KUKA KRL program: MyProgram_297().src

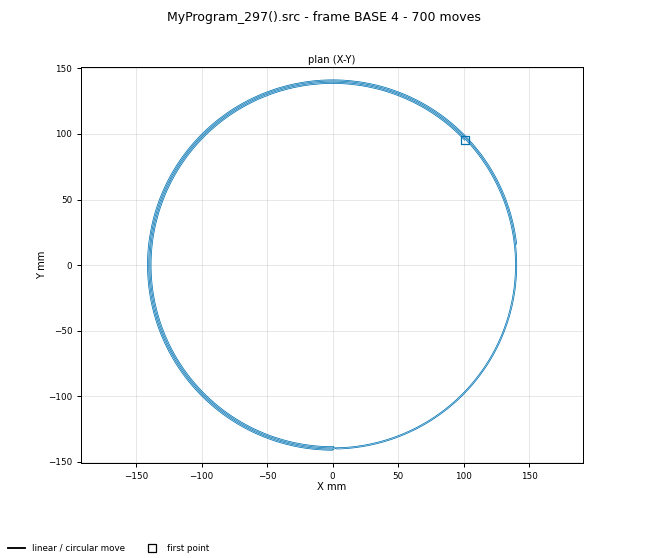
[picture p0: tool path of MyProgram_297().src in frame BASE 4, 700 of 700 moves have a stored position in this frame; points joined in program order, loops and branches not executed]
&ACCESS RVP
&REL 1
&PARAM TEMPLATE = C:\KRC\Roboter\Template\vorgabe
&PARAM EDITMASK = *
DEF MyProgram_297()
; ---- Setting reference (Base) ----
$BASE = BASE_DATA[4]

; --------------------------
; ---- Setting tool (TCP) ----
$TOOL = TOOL_DATA[3]
; --------------------------

$VEL.CP = VEL_APROX_PRINT
Startdeposition()
$VEL.CP = VEL_PRINT
LIN {X 100.7253,Y 95.1993,Z 178,A 45.1917,B 6.1181,C 0.1489,E1 6.2362,E2 407.2014} C_DIS
LIN {X 97.6837,Y 98.3177,Z 178,A 47.1151,B 6.1182,C 0.1434,E1 6.2323,E2 405.262} C_DIS
LIN {X 93.7907,Y 102.0381,Z 178,A 49.1623,B 6.1182,C 0.1418,E1 6.2282,E2 403.237} C_DIS
LIN {X 90.4705,Y 104.9931,Z 178,A 50.9851,B 6.1183,C 0.1386,E1 6.2244,E2 401.4158} C_DIS
LIN {X 87.1947,Y 107.7293,Z 178,A 52.6581,B 6.1183,C 0.1368,E1 6.2208,E2 399.754} C_DIS
LIN {X 83.9283,Y 110.2933,Z 178,A 54.4404,B 6.1185,C 0.1327,E1 6.2168,E2 397.9633} C_DIS
LIN {X 80.2806,Y 112.9764,Z 178,A 57.0009,B 6.1188,C 0.119,E1 6.2108,E2 395.3153} C_DIS
LIN {X 75.162,Y 116.444,Z 178,A 58.6179,B 6.1185,C 0.1293,E1 6.2073,E2 393.8171} C_DIS
LIN {X 71.7588,Y 118.5713,Z 178,A 60.415,B 6.1186,C 0.1247,E1 6.203,E2 392.0026} C_DIS
LIN {X 67.9906,Y 120.7715,Z 178,A 62.2218,B 6.1186,C 0.1221,E1 6.1986,E2 390.1954} C_DIS
LIN {X 64.2773,Y 122.7858,Z 178,A 63.932,B 6.1187,C 0.1203,E1 6.1944,E2 388.4897} C_DIS
LIN {X 60.7829,Y 124.554,Z 178,A 66.1002,B 6.1189,C 0.11,E1 6.1888,E2 386.2523} C_DIS
LIN {X 56.039,Y 126.7593,Z 178,A 67.8115,B 6.1189,C 0.1142,E1 6.1846,E2 384.5984} C_DIS
LIN {X 52.6665,Y 128.1983,Z 178,A 69.1021,B 6.1189,C 0.1158,E1 6.1813,E2 383.3363} C_DIS
LIN {X 50.1247,Y 129.2109,Z 178,A 70.2479,B 6.1189,C 0.1144,E1 6.1784,E2 382.1887} C_DIS
LIN {X 46.6313,Y 130.5129,Z 178,A 71.7515,B 6.1189,C 0.1134,E1 6.1744,E2 380.6901} C_DIS
LIN {X 43.0422,Y 131.7419,Z 178,A 73.3054,B 6.1189,C 0.1121,E1 6.1703,E2 379.1383} C_DIS
LIN {X 40.2799,Y 132.6106,Z 178,A 74.5276,B 6.1189,C 0.1107,E1 6.167,E2 377.9131} C_DIS
LIN {X 37.0505,Y 133.5489,Z 178,A 75.904,B 6.1189,C 0.1098,E1 6.1633,E2 376.5387} C_DIS
LIN {X 32.881,Y 134.6365,Z 178,A 77.8166,B 6.1189,C 0.1067,E1 6.1581,E2 374.6101} C_DIS
LIN {X 25.5972,Y 136.2093,Z 178,A 80.8088,B 6.1189,C 0.1061,E1 6.15,E2 371.6299} C_DIS
LIN {X 21.3585,Y 136.9374,Z 178,A 83.4736,B 6.1192,C 0.0929,E1 6.1423,E2 368.8539} C_DIS
LIN {X 14.2754,Y 137.857,Z 178,A 85.3447,B 6.119,C 0.1068,E1 6.1375,E2 367.1202} C_DIS
LIN {X 9.967,Y 138.2343,Z 178,A 87.2432,B 6.119,C 0.1048,E1 6.1322,E2 365.2086} C_DIS
LIN {X 6.2445,Y 138.4543,Z 178,A 88.9169,B 6.119,C 0.1028,E1 6.1275,E2 363.5191} C_DIS
LIN {X 1.7423,Y 138.5834,Z 178,A 90.7344,B 6.119,C 0.1032,E1 6.1224,E2 361.7079} C_DIS
LIN {X -2.2127,Y 138.5756,Z 178,A 92.2544,B 6.119,C 0.1048,E1 6.1182,E2 360.2029} C_DIS
LIN {X -5.8911,Y 138.4688,Z 178,A 93.7442,B 6.119,C 0.1053,E1 6.114,E2 358.7178} C_DIS
LIN {X -9.6122,Y 138.2602,Z 178,A 95.28,B 6.119,C 0.1056,E1 6.1098,E2 357.1834} C_DIS
LIN {X -18.0083,Y 137.4181,Z 178,A 98.4994,B 6.119,C 0.1101,E1 6.101,E2 353.9995} C_DIS
LIN {X -22.9135,Y 136.6857,Z 178,A 100.7104,B 6.119,C 0.1088,E1 6.0948,E2 351.7697} C_DIS
LIN {X -26.0665,Y 136.1196,Z 178,A 102.2509,B 6.119,C 0.1067,E1 6.0905,E2 350.2031} C_DIS
LIN {X -29.2745,Y 135.4658,Z 178,A 103.6444,B 6.119,C 0.107,E1 6.0866,E2 348.8054} C_DIS
LIN {X -33.7927,Y 134.4103,Z 178,A 105.6072,B 6.119,C 0.1077,E1 6.0813,E2 346.8383} C_DIS
LIN {X -37.8957,Y 133.3125,Z 178,A 107.194,B 6.119,C 0.1111,E1 6.0771,E2 345.2736} C_DIS
LIN {X -40.7847,Y 132.4561,Z 178,A 108.5376,B 6.119,C 0.1109,E1 6.0735,E2 343.9187} C_DIS
LIN {X -44.1224,Y 131.3822,Z 178,A 109.9811,B 6.1189,C 0.1122,E1 6.0696,E2 342.4769} C_DIS
LIN {X -48.0912,Y 129.9826,Z 178,A 111.7643,B 6.1189,C 0.1133,E1 6.0649,E2 340.6895} C_DIS
LIN {X -55.095,Y 127.171,Z 178,A 114.518,B 6.1187,C 0.1211,E1 6.058,E2 337.9836} C_DIS
LIN {X -58.8642,Y 125.4731,Z 178,A 116.9315,B 6.1188,C 0.1146,E1 6.0516,E2 335.4838} C_DIS
LIN {X -62.0184,Y 123.9445,Z 178,A 118.0563,B 6.1188,C 0.1203,E1 6.0489,E2 334.4006} C_DIS
LIN {X -64.646,Y 122.5922,Z 178,A 119.2808,B 6.1188,C 0.1219,E1 6.0459,E2 333.1766} C_DIS
LIN {X -68.3234,Y 120.5842,Z 178,A 121.1678,B 6.1187,C 0.1224,E1 6.0412,E2 331.2716} C_DIS
LIN {X -72.2248,Y 118.2883,Z 178,A 123.0723,B 6.1187,C 0.1248,E1 6.0366,E2 329.3644} C_DIS
LIN {X -76.1855,Y 115.7767,Z 178,A 125.0168,B 6.1186,C 0.1277,E1 6.0321,E2 327.4208} C_DIS
LIN {X -80.0632,Y 113.13,Z 178,A 127.0679,B 6.1186,C 0.1296,E1 6.0274,E2 325.3575} C_DIS
LIN {X -83.5881,Y 110.551,Z 178,A 128.8041,B 6.1185,C 0.1334,E1 6.0235,E2 323.6315} C_DIS
LIN {X -86.8755,Y 107.9868,Z 178,A 130.5701,B 6.1185,C 0.136,E1 6.0196,E2 321.8616} C_DIS
LIN {X -90.4313,Y 105.0269,Z 178,A 132.5625,B 6.1183,C 0.1386,E1 6.0154,E2 319.8609} C_DIS
LIN {X -94.299,Y 101.5687,Z 178,A 134.5455,B 6.1183,C 0.1446,E1 6.0113,E2 317.8999} C_DIS
LIN {X -97.1107,Y 98.8837,Z 178,A 136.3105,B 6.1182,C 0.146,E1 6.0077,E2 316.1166} C_DIS
LIN {X -100.4054,Y 95.537,Z 178,A 138.3895,B 6.1182,C 0.1484,E1 6.0037,E2 314.0221} C_DIS
LIN {X -103.4582,Y 92.2224,Z 178,A 140.1155,B 6.118,C 0.1539,E1 6.0005,E2 312.3149} C_DIS
LIN {X -106.0375,Y 89.2444,Z 178,A 141.7656,B 6.1179,C 0.1572,E1 5.9975,E2 310.6635} C_DIS
LIN {X -108.3675,Y 86.4,Z 178,A 143.3929,B 6.1179,C 0.1594,E1 5.9946,E2 309.0241} C_DIS
LIN {X -111.3703,Y 82.4939,Z 178,A 145.4041,B 6.1177,C 0.1643,E1 5.9912,E2 307.018} C_DIS
LIN {X -113.712,Y 79.2342,Z 178,A 147.1609,B 6.1177,C 0.1671,E1 5.9884,E2 305.2505} C_DIS
LIN {X -116.3293,Y 75.3392,Z 178,A 149.1049,B 6.1175,C 0.1717,E1 5.9854,E2 303.3076} C_DIS
LIN {X -118.5224,Y 71.8397,Z 178,A 150.8723,B 6.1175,C 0.1752,E1 5.9828,E2 301.5343} C_DIS
LIN {X -120.7551,Y 68.0198,Z 178,A 152.7493,B 6.1173,C 0.1793,E1 5.9802,E2 299.6529} C_DIS
LIN {X -123.7351,Y 62.4322,Z 178,A 155.3187,B 6.1171,C 0.1864,E1 5.9768,E2 297.092} C_DIS
LIN {X -125.4863,Y 58.8358,Z 178,A 156.9727,B 6.117,C 0.1907,E1 5.9748,E2 295.4395} C_DIS
LIN {X -126.4956,Y 56.6285,Z 178,A 158.0829,B 6.117,C 0.1922,E1 5.9736,E2 294.3167} C_DIS
LIN {X -127.9618,Y 53.2329,Z 178,A 160.2866,B 6.117,C 0.1891,E1 5.9711,E2 292.0288} C_DIS
LIN {X -129.9199,Y 48.2586,Z 178,A 162.2344,B 6.1167,C 0.1978,E1 5.9692,E2 290.1164} C_DIS
LIN {X -131.1832,Y 44.7149,Z 178,A 163.4264,B 6.1165,C 0.2058,E1 5.9682,E2 288.972} C_DIS
LIN {X -132.0421,Y 42.1053,Z 178,A 164.6413,B 6.1164,C 0.2081,E1 5.9671,E2 287.748} C_DIS
LIN {X -133.1106,Y 38.5962,Z 178,A 166.1683,B 6.1162,C 0.2121,E1 5.9659,E2 286.2209} C_DIS
LIN {X -134.175,Y 34.7196,Z 178,A 167.7959,B 6.1161,C 0.2171,E1 5.9648,E2 284.5993} C_DIS
LIN {X -134.8127,Y 32.1502,Z 178,A 168.9852,B 6.1161,C 0.2192,E1 5.964,E2 283.3989} C_DIS
LIN {X -135.5798,Y 28.7468,Z 178,A 170.8753,B 6.1161,C 0.2185,E1 5.9628,E2 281.4531} C_DIS
LIN {X -136.3289,Y 24.9548,Z 178,A 171.9926,B 6.1157,C 0.228,E1 5.9623,E2 280.3983} C_DIS
LIN {X -137.035,Y 20.7283,Z 178,A 173.8658,B 6.1155,C 0.232,E1 5.9614,E2 278.5138} C_DIS
LIN {X -137.4731,Y 17.5883,Z 178,A 175.2734,B 6.1155,C 0.2347,E1 5.9609,E2 277.0949} C_DIS
LIN {X -138.0078,Y 12.7341,Z 178,A 177.5784,B 6.1153,C 0.2374,E1 5.9603,E2 274.7552} C_DIS
LIN {X -138.3575,Y 8.0894,Z 178,A 179.3067,B 6.115,C 0.245,E1 5.9599,E2 273.0537} C_DIS
LIN {X -138.5482,Y 3.5444,Z 178,A -178.763,B 6.1148,C 0.2499,E1 5.9597,E2 271.1185} C_DIS
LIN {X -138.588,Y -1.3629,Z 178,A -176.4182,B 6.1148,C 0.2524,E1 5.9597,E2 268.7351} C_DIS
LIN {X -138.4345,Y -6.6374,Z 178,A -174.403,B 6.1144,C 0.2603,E1 5.96,E2 266.7428} C_DIS
LIN {X -138.1855,Y -10.6361,Z 178,A -172.6569,B 6.1142,C 0.2641,E1 5.9603,E2 264.9864} C_DIS
LIN {X -137.7888,Y -14.9093,Z 178,A -170.8181,B 6.114,C 0.2684,E1 5.9608,E2 263.1406} C_DIS
LIN {X -137.3126,Y -18.8119,Z 178,A -169.1039,B 6.1139,C 0.2721,E1 5.9615,E2 261.4163} C_DIS
LIN {X -136.7527,Y -22.5121,Z 178,A -167.6567,B 6.1136,C 0.2775,E1 5.9621,E2 259.983} C_DIS
LIN {X -136.1286,Y -26.0195,Z 178,A -166.1799,B 6.1135,C 0.2816,E1 5.9628,E2 258.5067} C_DIS
LIN {X -135.4008,Y -29.5757,Z 178,A -164.6551,B 6.1133,C 0.2855,E1 5.9637,E2 256.9798} C_DIS
LIN {X -134.6153,Y -32.9689,Z 178,A -163.1742,B 6.1131,C 0.289,E1 5.9647,E2 255.4947} C_DIS
LIN {X -133.8465,Y -35.9606,Z 178,A -161.9285,B 6.1129,C 0.2929,E1 5.9656,E2 254.2538} C_DIS
LIN {X -133.0131,Y -38.9292,Z 178,A -160.4892,B 6.1129,C 0.2946,E1 5.9667,E2 252.7941} C_DIS
LIN {X -131.8935,Y -42.5703,Z 178,A -158.855,B 6.1127,C 0.2982,E1 5.9681,E2 251.1534} C_DIS
LIN {X -130.1182,Y -47.7261,Z 178,A -156.6629,B 6.1123,C 0.3049,E1 5.9701,E2 248.9706} C_DIS
LIN {X -128.9024,Y -50.9183,Z 178,A -155.2152,B 6.1122,C 0.3082,E1 5.9716,E2 247.5191} C_DIS
LIN {X -127.6594,Y -53.9569,Z 178,A -153.8291,B 6.112,C 0.3115,E1 5.9731,E2 246.1301} C_DIS
LIN {X -126.4571,Y -56.7145,Z 178,A -152.4951,B 6.1119,C 0.3137,E1 5.9746,E2 244.7851} C_DIS
LIN {X -124.9377,Y -59.988,Z 178,A -150.9958,B 6.1117,C 0.3174,E1 5.9764,E2 243.2856} C_DIS
LIN {X -123.1323,Y -63.6163,Z 178,A -148.8755,B 6.1117,C 0.3167,E1 5.9792,E2 241.1085} C_DIS
LIN {X -121.2539,Y -67.1265,Z 178,A -147.9414,B 6.1111,C 0.3287,E1 5.9803,E2 240.2674} C_DIS
LIN {X -118.7782,Y -71.4166,Z 178,A -145.3999,B 6.1111,C 0.3281,E1 5.9839,E2 237.663} C_DIS
LIN {X -116.3136,Y -75.3634,Z 178,A -143.4433,B 6.1109,C 0.3323,E1 5.9869,E2 235.703} C_DIS
LIN {X -113.931,Y -78.9194,Z 178,A -141.6395,B 6.1107,C 0.336,E1 5.9897,E2 233.8955} C_DIS
LIN {X -111.2363,Y -82.6739,Z 178,A -139.711,B 6.1105,C 0.3401,E1 5.9929,E2 231.9653} C_DIS
LIN {X -108.3847,Y -86.3785,Z 178,A -137.7678,B 6.1103,C 0.3442,E1 5.9963,E2 230.0215} C_DIS
LIN {X -105.5981,Y -89.7636,Z 178,A -135.914,B 6.1101,C 0.3476,E1 5.9996,E2 228.1629} C_DIS
LIN {X -102.6518,Y -93.1187,Z 178,A -134.0717,B 6.1098,C 0.3515,E1 6.003,E2 226.3216} C_DIS
LIN {X -99.832,Y -96.1362,Z 178,A -132.2581,B 6.1098,C 0.3536,E1 6.0065,E2 224.4945} C_DIS
LIN {X -96.606,Y -99.3772,Z 178,A -130.4005,B 6.1095,C 0.3577,E1 6.0102,E2 222.6417} C_DIS
LIN {X -93.4399,Y -102.3603,Z 178,A -128.5488,B 6.1093,C 0.3604,E1 6.014,E2 220.7834} C_DIS
LIN {X -90.146,Y -105.2726,Z 178,A -126.6642,B 6.1092,C 0.3629,E1 6.018,E2 218.8903} C_DIS
LIN {X -86.5888,Y -108.2173,Z 178,A -124.7614,B 6.109,C 0.3662,E1 6.0221,E2 216.9886} C_DIS
LIN {X -83.0471,Y -110.9584,Z 178,A -122.3531,B 6.1092,C 0.3625,E1 6.0277,E2 214.5073} C_DIS
LIN {X -78.8969,Y -113.9467,Z 178,A -120.9727,B 6.1085,C 0.3748,E1 6.0306,E2 213.2236} C_DIS
LIN {X -76.2379,Y -115.7422,Z 178,A -119.2641,B 6.1086,C 0.372,E1 6.0347,E2 211.465} C_DIS
LIN {X -71.9067,Y -118.4818,Z 178,A -117.2397,B 6.1084,C 0.3762,E1 6.0395,E2 209.453} C_DIS
LIN {X -67.9145,Y -120.8143,Z 178,A -115.3273,B 6.1082,C 0.3787,E1 6.0441,E2 207.5406} C_DIS
LIN {X -63.9131,Y -122.9771,Z 178,A -112.8863,B 6.1085,C 0.3739,E1 6.0503,E2 205.0255} C_DIS
LIN {X -59.3138,Y -125.2598,Z 178,A -111.7959,B 6.1076,C 0.3895,E1 6.0527,E2 204.0707} C_DIS
LIN {X -55.6661,Y -126.9241,Z 178,A -109.7533,B 6.1077,C 0.3864,E1 6.0581,E2 201.9778} C_DIS
LIN {X -52.0497,Y -128.4477,Z 178,A -108.0497,B 6.1077,C 0.3869,E1 6.0625,E2 200.2632} C_DIS
LIN {X -48.7938,Y -129.7195,Z 178,A -106.5077,B 6.1077,C 0.3869,E1 6.0665,E2 198.7082} C_DIS
LIN {X -45.3055,Y -130.9785,Z 178,A -105.0417,B 6.1076,C 0.3891,E1 6.0704,E2 197.2509} C_DIS
LIN {X -41.5118,Y -132.2316,Z 178,A -103.4267,B 6.1075,C 0.3909,E1 6.0747,E2 195.6404} C_DIS
LIN {X -38.64,Y -133.0978,Z 178,A -102.1278,B 6.1075,C 0.3909,E1 6.0782,E2 194.3334} C_DIS
LIN {X -33.1805,Y -134.5643,Z 178,A -99.0562,B 6.108,C 0.3825,E1 6.0867,E2 191.164} C_DIS
LIN {X -27.5769,Y -135.8216,Z 178,A -97.6586,B 6.1071,C 0.3968,E1 6.0902,E2 189.8949} C_DIS
LIN {X -21.1122,Y -136.9755,Z 178,A -94.6575,B 6.1073,C 0.3939,E1 6.0986,E2 186.8554} C_DIS
LIN {X -17.645,Y -137.4657,Z 178,A -93.3149,B 6.1072,C 0.3958,E1 6.1023,E2 185.5262} C_DIS
LIN {X -14.6413,Y -137.8176,Z 178,A -91.9734,B 6.1072,C 0.3947,E1 6.106,E2 184.1721} C_DIS
LIN {X -10.2752,Y -138.2118,Z 178,A -90.1388,B 6.1072,C 0.3947,E1 6.1111,E2 182.3339} C_DIS
LIN {X -6.937,Y -138.4194,Z 178,A -88.7327,B 6.1072,C 0.3944,E1 6.1151,E2 180.9242} C_DIS
LIN {X -3.2907,Y -138.5553,Z 178,A -87.2392,B 6.1072,C 0.3945,E1 6.1192,E2 179.4319} C_DIS
LIN {X 1.0123,Y -138.5881,Z 178,A -85.629,B 6.1071,C 0.3967,E1 6.1237,E2 177.8431} C_DIS
Enddeposition()
LIN {X 1.0123,Y -138.5881,Z 178,A -85.629,B 6.1071,C 0.3967,E1 6.1237,E2 177.8431} C_DIS
Startdeposition()
$VEL.CP = VEL_PRINT
LIN {X 0.3223,Y -139.4978,Z 178,A -86.4941,B 6.0436,C 0.4078,E1 6.0583,E2 178.8356} C_DIS
LIN {X -3.5454,Y -139.4527,Z 178,A -87.9992,B 6.0436,C 0.4067,E1 6.0541,E2 180.3305} C_DIS
LIN {X -7.1717,Y -139.313,Z 178,A -89.4579,B 6.0437,C 0.4063,E1 6.05,E2 181.7857} C_DIS
LIN {X -10.8678,Y -139.0752,Z 178,A -91.0003,B 6.0437,C 0.4064,E1 6.0457,E2 183.3315} C_DIS
LIN {X -14.386,Y -138.7546,Z 178,A -92.4328,B 6.0437,C 0.406,E1 6.0417,E2 184.7622} C_DIS
LIN {X -18.0156,Y -138.3291,Z 178,A -93.9271,B 6.0437,C 0.4055,E1 6.0376,E2 186.2561} C_DIS
LIN {X -21.615,Y -137.8127,Z 178,A -95.4504,B 6.0437,C 0.4055,E1 6.0334,E2 187.7838} C_DIS
LIN {X -26.509,Y -136.9556,Z 178,A -97.5705,B 6.0437,C 0.4057,E1 6.0275,E2 189.915} C_DIS
LIN {X -31.0309,Y -136.0019,Z 178,A -99.4007,B 6.0439,C 0.4039,E1 6.0225,E2 191.7368} C_DIS
LIN {X -35.1536,Y -134.997,Z 178,A -101.3758,B 6.0437,C 0.4059,E1 6.0171,E2 193.7428} C_DIS
LIN {X -40.222,Y -133.5739,Z 178,A -103.4323,B 6.0439,C 0.4031,E1 6.0116,E2 195.7859} C_DIS
LIN {X -44.3434,Y -132.2617,Z 178,A -105.0412,B 6.0442,C 0.3996,E1 6.0074,E2 197.3732} C_DIS
LIN {X -47.3233,Y -131.2246,Z 178,A -106.5007,B 6.0441,C 0.4006,E1 6.0035,E2 198.8544} C_DIS
LIN {X -51.8194,Y -129.5155,Z 178,A -108.3865,B 6.0443,C 0.3976,E1 5.9986,E2 200.7287} C_DIS
LIN {X -54.7237,Y -128.3167,Z 178,A -109.8416,B 6.0443,C 0.3984,E1 5.9948,E2 202.2056} C_DIS
LIN {X -58.9864,Y -126.4129,Z 178,A -111.6098,B 6.0445,C 0.3944,E1 5.9904,E2 203.9543} C_DIS
LIN {X -62.6068,Y -124.6596,Z 178,A -113.4277,B 6.0445,C 0.3946,E1 5.9858,E2 205.7941} C_DIS
LIN {X -66.4871,Y -122.6357,Z 178,A -115.242,B 6.0446,C 0.3926,E1 5.9813,E2 207.6107} C_DIS
LIN {X -70.5308,Y -120.3551,Z 178,A -117.1397,B 6.0448,C 0.3899,E1 5.9767,E2 209.5071} C_DIS
LIN {X -74.4572,Y -117.9663,Z 178,A -118.9485,B 6.045,C 0.3863,E1 5.9724,E2 211.3056} C_DIS
LIN {X -77.8084,Y -115.7841,Z 178,A -120.8356,B 6.045,C 0.3868,E1 5.968,E2 213.2245} C_DIS
LIN {X -83.4625,Y -111.7764,Z 178,A -123.5507,B 6.0454,C 0.3808,E1 5.9619,E2 215.9223} C_DIS
LIN {X -86.935,Y -109.0974,Z 178,A -125.404,B 6.0455,C 0.3784,E1 5.9578,E2 217.782} C_DIS
LIN {X -90.4421,Y -106.2081,Z 178,A -127.2994,B 6.0457,C 0.3754,E1 5.9537,E2 219.6809} C_DIS
LIN {X -93.8098,Y -103.2456,Z 178,A -129.1509,B 6.0459,C 0.3722,E1 5.9498,E2 221.5333} C_DIS
LIN {X -97.0198,Y -100.2351,Z 178,A -130.9882,B 6.0461,C 0.3691,E1 5.9461,E2 223.3741} C_DIS
LIN {X -100.0855,Y -97.1744,Z 178,A -132.8486,B 6.0462,C 0.3665,E1 5.9424,E2 225.2445} C_DIS
LIN {X -103.3151,Y -93.7332,Z 178,A -134.7654,B 6.0465,C 0.3624,E1 5.9388,E2 227.158} C_DIS
LIN {X -106.1489,Y -90.5118,Z 178,A -136.5955,B 6.0467,C 0.3594,E1 5.9355,E2 228.9964} C_DIS
LIN {X -108.9179,Y -87.1606,Z 178,A -138.4497,B 6.0468,C 0.3564,E1 5.9322,E2 230.8589} C_DIS
LIN {X -111.7183,Y -83.5405,Z 178,A -140.3561,B 6.0471,C 0.3525,E1 5.9289,E2 232.7681} C_DIS
LIN {X -114.4517,Y -79.7544,Z 178,A -142.2746,B 6.0473,C 0.3481,E1 5.9258,E2 234.686} C_DIS
LIN {X -116.2615,Y -77.0934,Z 178,A -143.7509,B 6.0473,C 0.3468,E1 5.9235,E2 236.1817} C_DIS
LIN {X -118.9476,Y -72.8794,Z 178,A -145.6851,B 6.0477,C 0.3406,E1 5.9207,E2 238.0996} C_DIS
LIN {X -120.3674,Y -70.51,Z 178,A -147.2646,B 6.0477,C 0.3427,E1 5.9184,E2 239.7359} C_DIS
LIN {X -122.4618,Y -66.8059,Z 178,A -148.8201,B 6.048,C 0.3363,E1 5.9163,E2 241.2659} C_DIS
LIN {X -124.8761,Y -62.1739,Z 178,A -150.8063,B 6.0484,C 0.3292,E1 5.9138,E2 243.2305} C_DIS
LIN {X -126.4932,Y -58.8126,Z 178,A -152.5062,B 6.0484,C 0.3271,E1 5.9118,E2 244.9512} C_DIS
LIN {X -128.5303,Y -54.2179,Z 178,A -154.363,B 6.0489,C 0.3196,E1 5.9097,E2 246.7802} C_DIS
LIN {X -129.8442,Y -50.9913,Z 178,A -156.0907,B 6.0489,C 0.319,E1 5.9079,E2 248.5452} C_DIS
LIN {X -131.9966,Y -45.1295,Z 178,A -158.5339,B 6.0493,C 0.3108,E1 5.9056,E2 250.9713} C_DIS
LIN {X -133.1589,Y -41.5781,Z 178,A -160.1436,B 6.0495,C 0.3075,E1 5.9042,E2 252.5897} C_DIS
LIN {X -134.1836,Y -38.1385,Z 178,A -161.6845,B 6.0497,C 0.3042,E1 5.903,E2 254.1382} C_DIS
LIN {X -135.1933,Y -34.3833,Z 178,A -163.248,B 6.0499,C 0.2994,E1 5.9019,E2 255.6963} C_DIS
LIN {X -135.975,Y -31.149,Z 178,A -164.651,B 6.0501,C 0.296,E1 5.901,E2 257.1031} C_DIS
LIN {X -136.7965,Y -27.3206,Z 178,A -166.3624,B 6.0503,C 0.2926,E1 5.9001,E2 258.8265} C_DIS
LIN {X -137.5642,Y -23.1428,Z 178,A -167.8976,B 6.0506,C 0.2856,E1 5.8993,E2 260.3337} C_DIS
LIN {X -138.0283,Y -20.1962,Z 178,A -169.3041,B 6.0506,C 0.284,E1 5.8987,E2 261.7625} C_DIS
LIN {X -138.5928,Y -15.8732,Z 178,A -171.649,B 6.0506,C 0.2847,E1 5.8979,E2 264.1765} C_DIS
LIN {X -139.0057,Y -11.701,Z 178,A -172.9455,B 6.0511,C 0.2754,E1 5.8976,E2 265.4177} C_DIS
LIN {X -139.2898,Y -7.6336,Z 178,A -175.258,B 6.051,C 0.2772,E1 5.8972,E2 267.8098} C_DIS
LIN {X -139.4717,Y -2.7059,Z 178,A -177.3632,B 6.0512,C 0.2722,E1 5.8972,E2 269.9234} C_DIS
LIN {X -139.4768,Y 2.4022,Z 178,A -178.8572,B 6.0517,C 0.26,E1 5.8972,E2 271.3395} C_DIS
LIN {X -139.365,Y 6.1135,Z 178,A 178.8526,B 6.0516,C 0.2635,E1 5.8975,E2 273.725} C_DIS
LIN {X -139.0193,Y 11.54,Z 178,A 176.7976,B 6.0519,C 0.2553,E1 5.8979,E2 275.7558} C_DIS
LIN {X -138.5925,Y 15.8752,Z 178,A 175.3404,B 6.0523,C 0.2468,E1 5.8983,E2 277.1697} C_DIS
LIN {X -138.1322,Y 19.4689,Z 178,A 173.8745,B 6.0525,C 0.2424,E1 5.8989,E2 278.6316} C_DIS
LIN {X -137.5997,Y 22.9302,Z 178,A 172.3164,B 6.0525,C 0.2395,E1 5.8996,E2 280.2035} C_DIS
LIN {X -136.4381,Y 29.0561,Z 178,A 169.918,B 6.0529,C 0.2307,E1 5.9009,E2 282.5792} C_DIS
LIN {X -135.7528,Y 32.1087,Z 178,A 168.4295,B 6.0529,C 0.2292,E1 5.9018,E2 284.0923} C_DIS
LIN {X -134.7915,Y 35.926,Z 178,A 166.852,B 6.0532,C 0.2243,E1 5.9029,E2 285.6634} C_DIS
LIN {X -134.0376,Y 38.6482,Z 178,A 165.6447,B 6.0532,C 0.2216,E1 5.9038,E2 286.8756} C_DIS
LIN {X -132.9994,Y 42.0799,Z 178,A 164.0526,B 6.0534,C 0.2188,E1 5.9051,E2 288.4815} C_DIS
LIN {X -131.9971,Y 45.1279,Z 178,A 162.9028,B 6.0535,C 0.2135,E1 5.9061,E2 289.609} C_DIS
LIN {X -130.7766,Y 48.5494,Z 178,A 161.4479,B 6.0537,C 0.2091,E1 5.9075,E2 291.0579} C_DIS
LIN {X -129.7175,Y 51.3141,Z 178,A 159.7641,B 6.0537,C 0.2107,E1 5.9093,E2 292.7993} C_DIS
LIN {X -127.6546,Y 56.2518,Z 178,A 157.6571,B 6.0539,C 0.204,E1 5.9116,E2 294.893} C_DIS
LIN {X -126.1299,Y 59.5901,Z 178,A 156.3412,B 6.0541,C 0.1981,E1 5.9131,E2 296.1835} C_DIS
LIN {X -124.2884,Y 63.3384,Z 178,A 154.1697,B 6.0541,C 0.1984,E1 5.9159,E2 298.4105} C_DIS
LIN {X -122.6034,Y 66.5464,Z 178,A 152.8451,B 6.0542,C 0.193,E1 5.9176,E2 299.7134} C_DIS
LIN {X -120.4136,Y 70.4314,Z 178,A 150.9757,B 6.0544,C 0.1888,E1 5.9202,E2 301.5859} C_DIS
LIN {X -117.9566,Y 74.4727,Z 178,A 149.0545,B 6.0545,C 0.1839,E1 5.923,E2 303.5026} C_DIS
LIN {X -115.5646,Y 78.133,Z 178,A 147.2061,B 6.0546,C 0.1801,E1 5.9259,E2 305.356} C_DIS
LIN {X -113.0534,Y 81.7244,Z 178,A 145.4324,B 6.0548,C 0.1757,E1 5.9288,E2 307.1248} C_DIS
LIN {X -109.9842,Y 85.8114,Z 178,A 143.179,B 6.0548,C 0.1726,E1 5.9326,E2 309.3956} C_DIS
LIN {X -107.16,Y 89.3133,Z 178,A 141.3302,B 6.055,C 0.1685,E1 5.9359,E2 311.2429} C_DIS
LIN {X -103.6159,Y 93.4013,Z 178,A 138.6156,B 6.055,C 0.1691,E1 5.941,E2 314.0166} C_DIS
LIN {X -100.4507,Y 96.7971,Z 178,A 137.0856,B 6.0552,C 0.161,E1 5.9439,E2 315.4983} C_DIS
LIN {X -97.3979,Y 99.8686,Z 178,A 134.8234,B 6.0552,C 0.1628,E1 5.9485,E2 317.8188} C_DIS
LIN {X -93.8656,Y 103.195,Z 178,A 132.8703,B 6.0552,C 0.1585,E1 5.9525,E2 319.7653} C_DIS
LIN {X -90.4971,Y 106.1613,Z 178,A 131.396,B 6.0554,C 0.151,E1 5.9556,E2 321.1923} C_DIS
LIN {X -86.4274,Y 109.5004,Z 178,A 129.0822,B 6.0554,C 0.1488,E1 5.9606,E2 323.5231} C_DIS
LIN {X -80.5402,Y 113.9001,Z 178,A 126.1633,B 6.0556,C 0.1427,E1 5.9672,E2 326.4272} C_DIS
LIN {X -76.9222,Y 116.3743,Z 178,A 124.3085,B 6.0556,C 0.1404,E1 5.9715,E2 328.2873} C_DIS
LIN {X -72.9661,Y 118.8944,Z 178,A 122.3976,B 6.0557,C 0.1373,E1 5.976,E2 330.1948} C_DIS
LIN {X -69.0331,Y 121.2204,Z 178,A 120.4994,B 6.0557,C 0.1349,E1 5.9806,E2 332.0941} C_DIS
LIN {X -65.2642,Y 123.2889,Z 178,A 118.7277,B 6.0559,C 0.1326,E1 5.9849,E2 333.8652} C_DIS
LIN {X -62.4865,Y 124.7219,Z 178,A 117.2552,B 6.0559,C 0.1332,E1 5.9887,E2 335.3602} C_DIS
LIN {X -57.55,Y 127.074,Z 178,A 115.2692,B 6.0559,C 0.1275,E1 5.9936,E2 337.3123} C_DIS
LIN {X -52.8703,Y 129.0919,Z 178,A 112.7558,B 6.0559,C 0.1302,E1 6.0002,E2 339.8763} C_DIS
LIN {X -49.5221,Y 130.4123,Z 178,A 111.5938,B 6.056,C 0.1249,E1 6.0031,E2 340.9981} C_DIS
LIN {X -45.9172,Y 131.7235,Z 178,A 110.043,B 6.056,C 0.1231,E1 6.0072,E2 342.5447} C_DIS
LIN {X -42.5902,Y 132.8364,Z 178,A 108.6703,B 6.056,C 0.1211,E1 6.0108,E2 343.9079} C_DIS
LIN {X -39.2866,Y 133.8506,Z 178,A 107.219,B 6.0561,C 0.1203,E1 6.0147,E2 345.3623} C_DIS
LIN {X -34.7857,Y 135.0912,Z 178,A 105.1925,B 6.0561,C 0.1203,E1 6.0202,E2 347.4011} C_DIS
LIN {X -31.2494,Y 135.952,Z 178,A 103.7489,B 6.0561,C 0.1187,E1 6.0241,E2 348.8374} C_DIS
LIN {X -27.7276,Y 136.7137,Z 178,A 102.1669,B 6.0561,C 0.1191,E1 6.0285,E2 350.4313} C_DIS
LIN {X -19.1379,Y 138.1795,Z 178,A 98.6078,B 6.0561,C 0.1173,E1 6.0383,E2 353.986} C_DIS
LIN {X -16,Y 138.5777,Z 178,A 96.7185,B 6.0561,C 0.1245,E1 6.0437,E2 355.9474} C_DIS
LIN {X -10.874,Y 139.0747,Z 178,A 95.1928,B 6.0561,C 0.1165,E1 6.0477,E2 357.3994} C_DIS
LIN {X -7.2758,Y 139.3078,Z 178,A 93.6835,B 6.0561,C 0.1166,E1 6.052,E2 358.9115} C_DIS
LIN {X -3.1172,Y 139.4647,Z 178,A 92.0375,B 6.0561,C 0.1157,E1 6.0565,E2 360.5488} C_DIS
LIN {X 0.0659,Y 139.4992,Z 178,A 90.6172,B 6.0561,C 0.1172,E1 6.0605,E2 361.9826} C_DIS
LIN {X 4.3313,Y 139.4309,Z 178,A 88.8827,B 6.0561,C 0.1172,E1 6.0654,E2 363.7141} C_DIS
LIN {X 8.6216,Y 139.2307,Z 178,A 87.2428,B 6.0561,C 0.1158,E1 6.0699,E2 365.3379} C_DIS
LIN {X 11.654,Y 139.0097,Z 178,A 85.8808,B 6.0561,C 0.1176,E1 6.0737,E2 366.7135} C_DIS
LIN {X 15.9985,Y 138.5778,Z 178,A 83.8576,B 6.0561,C 0.1213,E1 6.0794,E2 368.7645} C_DIS
LIN {X 19.3433,Y 138.1498,Z 178,A 82.3529,B 6.0561,C 0.1235,E1 6.0836,E2 370.2835} C_DIS
LIN {X 23.4661,Y 137.5103,Z 178,A 80.9891,B 6.0561,C 0.1196,E1 6.0873,E2 371.6036} C_DIS
LIN {X 26.497,Y 136.9579,Z 178,A 79.588,B 6.0561,C 0.1222,E1 6.0912,E2 373.0211} C_DIS
LIN {X 30.9568,Y 136.0189,Z 178,A 77.6366,B 6.0561,C 0.1245,E1 6.0965,E2 374.9819} C_DIS
LIN {X 34.3666,Y 135.1975,Z 178,A 76.5277,B 6.0561,C 0.1209,E1 6.0994,E2 376.0493} C_DIS
LIN {X 37.6745,Y 134.3133,Z 178,A 75.0789,B 6.0561,C 0.1226,E1 6.1033,E2 377.503} C_DIS
LIN {X 41.999,Y 133.0253,Z 178,A 73.2573,B 6.0561,C 0.1237,E1 6.1082,E2 379.3203} C_DIS
LIN {X 44.7765,Y 132.1174,Z 178,A 72.024,B 6.0561,C 0.1253,E1 6.1114,E2 380.5576} C_DIS
LIN {X 48.3767,Y 130.8413,Z 178,A 70.4818,B 6.056,C 0.1265,E1 6.1155,E2 382.0962} C_DIS
LIN {X 51.5318,Y 129.6315,Z 178,A 69.1032,B 6.056,C 0.1278,E1 6.1191,E2 383.4735} C_DIS
LIN {X 55.3446,Y 128.0482,Z 178,A 67.4845,B 6.056,C 0.1286,E1 6.1232,E2 385.0824} C_DIS
LIN {X 58.1626,Y 126.7938,Z 178,A 65.8892,B 6.0558,C 0.1349,E1 6.1274,E2 386.7185} C_DIS
LIN {X 61.4304,Y 125.2429,Z 178,A 64.9622,B 6.0559,C 0.1287,E1 6.1295,E2 387.5757} C_DIS
LIN {X 63.2352,Y 124.341,Z 178,A 63.7611,B 6.0558,C 0.1352,E1 6.1326,E2 388.8233} C_DIS
LIN {X 67.7011,Y 121.9693,Z 178,A 61.7992,B 6.0558,C 0.1364,E1 6.1374,E2 390.7709} C_DIS
LIN {X 71.6195,Y 119.7106,Z 178,A 59.9663,B 6.0558,C 0.1387,E1 6.1418,E2 392.6007} C_DIS
LIN {X 75.5459,Y 117.2728,Z 178,A 58.3342,B 6.0558,C 0.1377,E1 6.1456,E2 394.1996} C_DIS
LIN {X 78.8146,Y 115.1008,Z 178,A 56.431,B 6.0556,C 0.1446,E1 6.1501,E2 396.1394} C_DIS
LIN {X 82.9305,Y 112.1724,Z 178,A 54.4183,B 6.0556,C 0.1472,E1 6.1546,E2 398.1446} C_DIS
LIN {X 86.4771,Y 109.4614,Z 178,A 52.6482,B 6.0555,C 0.1495,E1 6.1585,E2 399.9069} C_DIS
LIN {X 89.9521,Y 106.624,Z 178,A 50.831,B 6.0554,C 0.1524,E1 6.1624,E2 401.7212} C_DIS
LIN {X 93.6146,Y 103.4227,Z 178,A 49.0313,B 6.0554,C 0.1532,E1 6.1661,E2 403.4963} C_DIS
LIN {X 98.191,Y 99.0883,Z 178,A 46.3028,B 6.0552,C 0.1605,E1 6.1717,E2 406.243} C_DIS
LIN {X 101.364,Y 95.8399,Z 178,A 44.4675,B 6.0551,C 0.1639,E1 6.1752,E2 408.0751} C_DIS
LIN {X 104.5693,Y 92.332,Z 178,A 42.6194,B 6.0551,C 0.1664,E1 6.1786,E2 409.9108} C_DIS
LIN {X 107.3343,Y 89.1028,Z 178,A 41.0208,B 6.055,C 0.1679,E1 6.1815,E2 411.4912} C_DIS
LIN {X 111.2162,Y 84.2077,Z 178,A 38.3519,B 6.0548,C 0.1753,E1 6.1861,E2 414.1741} C_DIS
LIN {X 113.7481,Y 80.7557,Z 178,A 36.6171,B 6.0547,C 0.179,E1 6.1889,E2 415.9066} C_DIS
LIN {X 115.9816,Y 77.5127,Z 178,A 35.0402,B 6.0546,C 0.1822,E1 6.1914,E2 417.4791} C_DIS
LIN {X 118.6188,Y 73.414,Z 178,A 32.6995,B 6.0543,C 0.1924,E1 6.1949,E2 419.8633} C_DIS
LIN {X 120.7811,Y 69.7976,Z 178,A 31.2223,B 6.0543,C 0.1926,E1 6.197,E2 421.3093} C_DIS
LIN {X 123.2989,Y 65.2453,Z 178,A 29.3158,B 6.0542,C 0.1943,E1 6.1995,E2 423.1877} C_DIS
LIN {X 125.0268,Y 61.8684,Z 178,A 28.0856,B 6.0542,C 0.1929,E1 6.201,E2 424.3769} C_DIS
LIN {X 126.6729,Y 58.4241,Z 178,A 26.3504,B 6.054,C 0.1997,E1 6.2031,E2 426.1343} C_DIS
LIN {X 127.9824,Y 55.4969,Z 178,A 24.5811,B 6.0537,C 0.2105,E1 6.2051,E2 427.9616} C_DIS
LIN {X 129.6204,Y 51.5592,Z 178,A 23.0061,B 6.0536,C 0.2122,E1 6.2067,E2 429.5154} C_DIS
LIN {X 130.8249,Y 48.4204,Z 178,A 21.8578,B 6.0536,C 0.2122,E1 6.2078,E2 430.6349} C_DIS
LIN {X 132.2634,Y 44.3381,Z 178,A 20.2393,B 6.0536,C 0.2143,E1 6.2093,E2 432.2342} C_DIS
LIN {X 133.3531,Y 40.9438,Z 178,A 18.8112,B 6.0534,C 0.2177,E1 6.2105,E2 433.6586} C_DIS
LIN {X 134.2807,Y 37.791,Z 178,A 17.5332,B 6.0534,C 0.2202,E1 6.2115,E2 434.9282} C_DIS
LIN {X 135.2106,Y 34.3151,Z 178,A 16.0446,B 6.0532,C 0.2245,E1 6.2125,E2 436.4192} C_DIS
LIN {X 136.2945,Y 29.7213,Z 178,A 13.9274,B 6.0528,C 0.2328,E1 6.2138,E2 438.5605} C_DIS
LIN {X 137.3794,Y 24.2179,Z 178,A 11.2694,B 6.0524,C 0.2451,E1 6.2152,E2 441.265} C_DIS
LIN {X 138.1843,Y 19.1044,Z 178,A 9.5224,B 6.0524,C 0.2449,E1 6.2159,E2 442.9655} C_DIS
LIN {X 138.5963,Y 15.8436,Z 178,A 8.4514,B 6.0524,C 0.2441,E1 6.2162,E2 444.0018} C_DIS
LIN {X 138.9346,Y 12.5422,Z 178,A 7.0101,B 6.0522,C 0.2493,E1 6.2166,E2 445.4542} C_DIS
LIN {X 139.2226,Y 8.753,Z 178,A 5.6448,B 6.0522,C 0.2504,E1 6.2168,E2 446.7955} C_DIS
LIN {X 139.3947,Y 5.3534,Z 178,A 4.2125,B 6.0519,C 0.255,E1 6.217,E2 448.2332} C_DIS
LIN {X 139.4948,Y 0.95,Z 178,A 2.5102,B 6.0519,C 0.2584,E1 6.2171,E2 449.9233} C_DIS
LIN {X 139.4711,Y -2.745,Z 178,A 0.8838,B 6.0515,C 0.2645,E1 6.2171,E2 451.5648} C_DIS
LIN {X 139.3334,Y -6.7652,Z 178,A -0.612,B 6.0515,C 0.2667,E1 6.2169,E2 453.0418} C_DIS
LIN {X 139.1135,Y -10.3423,Z 178,A -2.0793,B 6.0513,C 0.2708,E1 6.2166,E2 454.5098} C_DIS
LIN {X 138.7275,Y -14.6373,Z 178,A -3.8502,B 6.051,C 0.2758,E1 6.2161,E2 456.2821} C_DIS
LIN {X 138.2297,Y -18.7735,Z 178,A -5.5551,B 6.0508,C 0.2806,E1 6.2155,E2 457.9877} C_DIS
LIN {X 137.641,Y -22.6826,Z 178,A -6.9177,B 6.0508,C 0.2808,E1 6.2149,E2 459.3179} C_DIS
LIN {X 137.109,Y -25.7052,Z 178,A -8.4281,B 6.0504,C 0.2886,E1 6.2142,E2 460.8617} C_DIS
LIN {X 136.0964,Y -30.6173,Z 178,A -10.2564,B 6.0504,C 0.2905,E1 6.2131,E2 462.6619} C_DIS
LIN {X 135.413,Y -33.5178,Z 178,A -11.6469,B 6.0501,C 0.2967,E1 6.2122,E2 464.0751} C_DIS
LIN {X 133.8126,Y -39.4166,Z 178,A -14.1356,B 6.0497,C 0.3033,E1 6.2103,E2 466.5631} C_DIS
LIN {X 132.5547,Y -43.4634,Z 178,A -15.7447,B 6.0496,C 0.3059,E1 6.2089,E2 468.1568} C_DIS
LIN {X 131.3245,Y -47.0464,Z 178,A -17.1245,B 6.0496,C 0.3072,E1 6.2077,E2 469.5151} C_DIS
LIN {X 130.2915,Y -49.8407,Z 178,A -18.3637,B 6.0494,C 0.3107,E1 6.2065,E2 470.7575} C_DIS
LIN {X 128.9198,Y -53.2854,Z 178,A -19.7178,B 6.0493,C 0.312,E1 6.2051,E2 472.091} C_DIS
LIN {X 127.5588,Y -56.466,Z 178,A -21.2375,B 6.049,C 0.3174,E1 6.2034,E2 473.6248} C_DIS
LIN {X 125.9976,Y -59.8671,Z 178,A -22.8503,B 6.0487,C 0.3227,E1 6.2014,E2 475.2489} C_DIS
LIN {X 123.9794,Y -63.9454,Z 178,A -24.7005,B 6.0485,C 0.3272,E1 6.1991,E2 477.0985} C_DIS
LIN {X 121.741,Y -68.1113,Z 178,A -26.5681,B 6.0483,C 0.331,E1 6.1966,E2 478.9581} C_DIS
LIN {X 119.2584,Y -72.37,Z 178,A -28.8685,B 6.0478,C 0.3405,E1 6.1933,E2 481.2962} C_DIS
LIN {X 117.0724,Y -75.8552,Z 178,A -30.1616,B 6.0478,C 0.3382,E1 6.1914,E2 482.5393} C_DIS
LIN {X 114.6417,Y -79.4812,Z 178,A -31.7569,B 6.0478,C 0.3393,E1 6.1889,E2 484.1104} C_DIS
LIN {X 112.3212,Y -82.7279,Z 178,A -34.2934,B 6.0468,C 0.3577,E1 6.1845,E2 486.765} C_DIS
LIN {X 108.4098,Y -87.7914,Z 178,A -36.1341,B 6.0472,C 0.351,E1 6.1815,E2 488.506} C_DIS
LIN {X 106.0727,Y -90.6014,Z 178,A -37.6685,B 6.0469,C 0.355,E1 6.1787,E2 490.0462} C_DIS
LIN {X 103.8038,Y -93.1918,Z 178,A -39.0382,B 6.0468,C 0.3573,E1 6.1762,E2 491.4113} C_DIS
LIN {X 100.949,Y -96.277,Z 178,A -40.67,B 6.0467,C 0.3595,E1 6.1731,E2 493.0323} C_DIS
LIN {X 97.9374,Y -99.3394,Z 178,A -42.4233,B 6.0464,C 0.3631,E1 6.1696,E2 494.7858} C_DIS
LIN {X 94.7705,Y -102.3652,Z 178,A -44.0832,B 6.0464,C 0.3645,E1 6.1663,E2 496.4291} C_DIS
LIN {X 92.1261,Y -104.7503,Z 178,A -45.9474,B 6.0458,C 0.3738,E1 6.1623,E2 498.3471} C_DIS
LIN {X 89.0635,Y -107.3668,Z 178,A -47.2531,B 6.0459,C 0.3714,E1 6.1596,E2 499.6086} C_DIS
LIN {X 85.6663,Y -110.0967,Z 178,A -49.1406,B 6.0456,C 0.3763,E1 6.1554,E2 501.5105} C_DIS
LIN {X 82.4293,Y -112.5405,Z 178,A -50.6829,B 6.0456,C 0.3773,E1 6.152,E2 503.038} C_DIS
LIN {X 77.6576,Y -115.8848,Z 178,A -53.0427,B 6.0454,C 0.3809,E1 6.1466,E2 505.3954} C_DIS
LIN {X 75.0557,Y -117.5866,Z 178,A -54.4221,B 6.0451,C 0.3846,E1 6.1433,E2 506.7893} C_DIS
LIN {X 71.4841,Y -119.7913,Z 178,A -56.4906,B 6.0446,C 0.3926,E1 6.1382,E2 508.9043} C_DIS
LIN {X 67.075,Y -122.3151,Z 178,A -58.0768,B 6.0449,C 0.388,E1 6.1345,E2 510.4268} C_DIS
LIN {X 63.5594,Y -124.1759,Z 178,A -59.5128,B 6.0449,C 0.3873,E1 6.131,E2 511.838} C_DIS
LIN {X 60.4575,Y -125.7155,Z 178,A -60.9355,B 6.0449,C 0.3892,E1 6.1274,E2 513.2618} C_DIS
LIN {X 57.1842,Y -127.2376,Z 178,A -62.3826,B 6.0447,C 0.3906,E1 6.1238,E2 514.7054} C_DIS
LIN {X 54.253,Y -128.5157,Z 178,A -63.7152,B 6.0447,C 0.3925,E1 6.1203,E2 516.0416} C_DIS
LIN {X 51.0674,Y -129.8146,Z 178,A -65.1883,B 6.0444,C 0.3951,E1 6.1165,E2 517.5236} C_DIS
LIN {X 48.0525,Y -130.9617,Z 178,A -66.5255,B 6.0444,C 0.3967,E1 6.113,E2 518.8634} C_DIS
LIN {X 44.181,Y -132.3158,Z 178,A -68.1285,B 6.0444,C 0.3972,E1 6.1088,E2 520.4568} C_DIS
LIN {X 39.9244,Y -133.6639,Z 178,A -70.1726,B 6.044,C 0.4021,E1 6.1032,E2 522.5298} C_DIS
LIN {X 35.1362,Y -135.0021,Z 178,A -72.7236,B 6.0434,C 0.4113,E1 6.0962,E2 525.1487} C_DIS
LIN {X 29.5038,Y -136.3414,Z 178,A -74.1935,B 6.0441,C 0.3998,E1 6.0925,E2 526.5011} C_DIS
LIN {X 23.7282,Y -137.4665,Z 178,A -77.2141,B 6.0434,C 0.4101,E1 6.084,E2 529.6026} C_DIS
LIN {X 19.544,Y -138.1215,Z 178,A -78.538,B 6.0438,C 0.4051,E1 6.0804,E2 530.873} C_DIS
LIN {X 15.5375,Y -138.6307,Z 178,A -80.1306,B 6.0438,C 0.4049,E1 6.076,E2 532.4578} C_DIS
LIN {X 12.0827,Y -138.9735,Z 178,A -81.5932,B 6.0438,C 0.406,E1 6.072,E2 533.9261} C_DIS
LIN {X 8.2921,Y -139.251,Z 178,A -83.179,B 6.0437,C 0.4068,E1 6.0675,E2 535.5159} C_DIS
LIN {X 3.8826,Y -139.4434,Z 178,A -84.8943,B 6.0437,C 0.4059,E1 6.0628,E2 537.2193} C_DIS
LIN {X 1.0209,Y -139.4912,Z 178,A -85.6588,B 6.0441,C 0.4003,E1 6.0608,E2 537.93} C_DIS
Enddeposition()
LIN {X 1.0209,Y -139.4912,Z 178,A -85.6588,B 6.0441,C 0.4003,E1 6.0608,E2 537.93} C_DIS
Startdeposition()
$VEL.CP = VEL_PRINT
LIN {X 3.2449,Y -140.3657,Z 178,A -84.2836,B 5.8198,C 0.3947,E1 5.8403,E2 536.5889} C_DIS
LIN {X 7.3424,Y -140.2098,Z 178,A -82.6673,B 5.8198,C 0.3951,E1 5.8448,E2 534.9794} C_DIS
LIN {X 11.6841,Y -139.9146,Z 178,A -80.9787,B 5.8198,C 0.3957,E1 5.8495,E2 533.3015} C_DIS
LIN {X 15.6684,Y -139.526,Z 178,A -79.2201,B 5.8199,C 0.3933,E1 5.8544,E2 531.5254} C_DIS
LIN {X 22.3206,Y -138.6174,Z 178,A -76.5877,B 5.8199,C 0.3933,E1 5.8617,E2 528.9059} C_DIS
LIN {X 25.6691,Y -138.0368,Z 178,A -75.2992,B 5.8199,C 0.3939,E1 5.8652,E2 527.6297} C_DIS
LIN {X 29.8855,Y -137.1841,Z 178,A -73.0278,B 5.8205,C 0.3852,E1 5.8716,E2 525.2877} C_DIS
LIN {X 34.1479,Y -136.1859,Z 178,A -71.5666,B 5.8203,C 0.3885,E1 5.8754,E2 523.8693} C_DIS
LIN {X 38.7867,Y -134.939,Z 178,A -69.6538,B 5.8203,C 0.3874,E1 5.8805,E2 521.9616} C_DIS
LIN {X 42.9397,Y -133.674,Z 178,A -67.9948,B 5.8203,C 0.3874,E1 5.8849,E2 520.3165} C_DIS
LIN {X 46.2532,Y -132.564,Z 178,A -66.6019,B 5.8203,C 0.3864,E1 5.8886,E2 518.9271} C_DIS
LIN {X 49.9988,Y -131.1993,Z 178,A -65.0026,B 5.8205,C 0.385,E1 5.8928,E2 517.3303} C_DIS
LIN {X 53.2132,Y -129.9286,Z 178,A -63.6135,B 5.8205,C 0.3836,E1 5.8964,E2 515.943} C_DIS
LIN {X 56.3774,Y -128.5869,Z 178,A -62.2284,B 5.8207,C 0.3822,E1 5.8999,E2 514.5592} C_DIS
LIN {X 59.0999,Y -127.3566,Z 178,A -61.0055,B 5.8207,C 0.3805,E1 5.903,E2 513.3349} C_DIS
LIN {X 62.1415,Y -125.9003,Z 178,A -59.6103,B 5.8209,C 0.3784,E1 5.9065,E2 511.936} C_DIS
LIN {X 65.473,Y -124.2006,Z 178,A -58.1692,B 5.8209,C 0.3775,E1 5.9101,E2 510.5052} C_DIS
LIN {X 69.7063,Y -121.8774,Z 178,A -55.8954,B 5.8215,C 0.37,E1 5.9157,E2 508.1891} C_DIS
LIN {X 72.6364,Y -120.154,Z 178,A -54.3489,B 5.8217,C 0.3653,E1 5.9195,E2 506.62} C_DIS
LIN {X 76.3768,Y -117.8118,Z 178,A -53.0474,B 5.8214,C 0.3701,E1 5.9224,E2 505.3843} C_DIS
LIN {X 81.9919,Y -113.9754,Z 178,A -50.1968,B 5.8218,C 0.3641,E1 5.929,E2 502.5214} C_DIS
LIN {X 85.6019,Y -111.2901,Z 178,A -48.4659,B 5.8219,C 0.3625,E1 5.9328,E2 500.803} C_DIS
LIN {X 88.6362,Y -108.8885,Z 178,A -46.8373,B 5.8222,C 0.3587,E1 5.9363,E2 499.1664} C_DIS
LIN {X 93.393,Y -104.8375,Z 178,A -44.4636,B 5.8222,C 0.3565,E1 5.9413,E2 496.8141} C_DIS
LIN {X 96.2522,Y -102.2181,Z 178,A -42.8147,B 5.8225,C 0.3523,E1 5.9447,E2 495.1549} C_DIS
LIN {X 99.3207,Y -99.24,Z 178,A -41.1145,B 5.8227,C 0.3494,E1 5.9481,E2 493.4592} C_DIS
LIN {X 103.5194,Y -94.8515,Z 178,A -38.6335,B 5.823,C 0.344,E1 5.9528,E2 490.9757} C_DIS
LIN {X 106.6418,Y -91.3275,Z 178,A -36.7405,B 5.8233,C 0.3402,E1 5.9563,E2 489.0848} C_DIS
LIN {X 109.4745,Y -87.9116,Z 178,A -34.6372,B 5.8238,C 0.3314,E1 5.9601,E2 486.9405} C_DIS
LIN {X 112.0688,Y -84.579,Z 178,A -33.3004,B 5.8236,C 0.3336,E1 5.9622,E2 485.654} C_DIS
LIN {X 116.381,Y -78.5399,Z 178,A -30.5902,B 5.8238,C 0.3315,E1 5.9665,E2 482.9835} C_DIS
LIN {X 118.1116,Y -75.9127,Z 178,A -28.7381,B 5.8244,C 0.3192,E1 5.9695,E2 481.0545} C_DIS
LIN {X 120.3162,Y -72.3681,Z 178,A -27.4644,B 5.8243,C 0.3219,E1 5.9712,E2 479.8367} C_DIS
LIN {X 122.4864,Y -68.6306,Z 178,A -25.7002,B 5.8245,C 0.3175,E1 5.9737,E2 478.0707} C_DIS
LIN {X 124.7922,Y -64.3418,Z 178,A -23.6146,B 5.8249,C 0.3108,E1 5.9764,E2 475.9702} C_DIS
LIN {X 126.7614,Y -60.366,Z 178,A -22.0615,B 5.8249,C 0.3103,E1 5.9782,E2 474.4497} C_DIS
LIN {X 128.3514,Y -56.9087,Z 178,A -20.5556,B 5.8251,C 0.3069,E1 5.98,E2 472.9487} C_DIS
LIN {X 129.785,Y -53.5601,Z 178,A -19.0339,B 5.8253,C 0.3024,E1 5.9816,E2 471.421} C_DIS
LIN {X 130.9592,Y -50.6187,Z 178,A -17.7874,B 5.8255,C 0.2997,E1 5.9829,E2 470.1794} C_DIS
LIN {X 132.3672,Y -46.8204,Z 178,A -16.2112,B 5.8256,C 0.2965,E1 5.9844,E2 468.612} C_DIS
LIN {X 133.3807,Y -43.8449,Z 178,A -14.9772,B 5.8258,C 0.2938,E1 5.9855,E2 467.3832} C_DIS
LIN {X 134.6014,Y -39.9403,Z 178,A -12.9385,B 5.8263,C 0.2831,E1 5.9871,E2 465.294} C_DIS
LIN {X 135.6496,Y -36.2176,Z 178,A -11.1253,B 5.8267,C 0.2748,E1 5.9885,E2 463.448} C_DIS
LIN {X 136.9683,Y -30.8609,Z 178,A -9.7775,B 5.8263,C 0.2835,E1 5.9893,E2 462.2183} C_DIS
LIN {X 138.1086,Y -25.2757,Z 178,A -7.1794,B 5.8268,C 0.2724,E1 5.9907,E2 459.5824} C_DIS
LIN {X 138.7585,Y -21.4159,Z 178,A -5.6924,B 5.8269,C 0.2697,E1 5.9913,E2 458.1086} C_DIS
LIN {X 139.2414,Y -18.0126,Z 178,A -4.3646,B 5.8271,C 0.267,E1 5.9918,E2 456.7895} C_DIS
LIN {X 139.7375,Y -13.6409,Z 178,A -2.5413,B 5.8273,C 0.2614,E1 5.9923,E2 454.9611} C_DIS
LIN {X 140.0873,Y -9.4214,Z 178,A -0.7885,B 5.8276,C 0.2561,E1 5.9927,E2 453.2037} C_DIS
LIN {X 140.3005,Y -5.3303,Z 178,A 0.6842,B 5.8276,C 0.2546,E1 5.9929,E2 451.7557} C_DIS
LIN {X 140.3962,Y -1.4101,Z 178,A 2.3756,B 5.8279,C 0.2485,E1 5.9929,E2 450.0512} C_DIS
LIN {X 140.3787,Y 2.5468,Z 178,A 3.8313,B 5.8279,C 0.2465,E1 5.9929,E2 448.6151} C_DIS
LIN {X 140.2574,Y 6.3959,Z 178,A 5.478,B 5.8282,C 0.2408,E1 5.9927,E2 446.9574} C_DIS
LIN {X 140.0209,Y 10.3319,Z 178,A 6.9034,B 5.8282,C 0.2392,E1 5.9925,E2 445.5547} C_DIS
LIN {X 139.7017,Y 14.014,Z 178,A 8.3614,B 5.8284,C 0.2358,E1 5.9921,E2 444.1023} C_DIS
LIN {X 138.6984,Y 21.8039,Z 178,A 11.5107,B 5.8287,C 0.2277,E1 5.9909,E2 440.9582} C_DIS
LIN {X 138.0573,Y 25.5617,Z 178,A 13.0266,B 5.8289,C 0.224,E1 5.9902,E2 439.4465} C_DIS
LIN {X 137.4675,Y 28.5582,Z 178,A 14.2482,B 5.8289,C 0.2209,E1 5.9895,E2 438.2272} C_DIS
LIN {X 136.7333,Y 31.8897,Z 178,A 15.7433,B 5.8292,C 0.2153,E1 5.9886,E2 436.7178} C_DIS
LIN {X 135.7647,Y 35.7859,Z 178,A 17.3211,B 5.8293,C 0.2118,E1 5.9875,E2 435.1468} C_DIS
LIN {X 134.671,Y 39.7027,Z 178,A 18.8451,B 5.8294,C 0.2094,E1 5.9863,E2 433.6394} C_DIS
LIN {X 133.7026,Y 42.8502,Z 178,A 20.1867,B 5.8295,C 0.2058,E1 5.9852,E2 432.2973} C_DIS
LIN {X 132.4335,Y 46.6297,Z 178,A 21.7335,B 5.8296,C 0.2027,E1 5.9838,E2 430.76} C_DIS
LIN {X 131.4283,Y 49.3872,Z 178,A 23.4804,B 5.8301,C 0.1907,E1 5.982,E2 428.9407} C_DIS
LIN {X 129.6084,Y 53.9829,Z 178,A 24.6291,B 5.8298,C 0.1994,E1 5.9809,E2 427.904} C_DIS
LIN {X 128.6787,Y 56.1648,Z 178,A 25.7678,B 5.8299,C 0.1941,E1 5.9796,E2 426.7427} C_DIS
LIN {X 127.4882,Y 58.8153,Z 178,A 26.9975,B 5.8301,C 0.1903,E1 5.9782,E2 425.5066} C_DIS
LIN {X 125.5732,Y 62.8046,Z 178,A 28.7574,B 5.8301,C 0.1864,E1 5.976,E2 423.7519} C_DIS
LIN {X 123.9303,Y 65.9878,Z 178,A 30.2668,B 5.8303,C 0.182,E1 5.9741,E2 422.2357} C_DIS
LIN {X 120.5304,Y 72.0102,Z 178,A 33.0584,B 5.8305,C 0.1755,E1 5.9702,E2 419.4468} C_DIS
LIN {X 118.1148,Y 75.9077,Z 178,A 34.8829,B 5.8306,C 0.1717,E1 5.9675,E2 417.6276} C_DIS
LIN {X 115.7549,Y 79.4597,Z 178,A 36.5773,B 5.8307,C 0.1683,E1 5.9648,E2 415.9384} C_DIS
LIN {X 113.2403,Y 83.0041,Z 178,A 38.288,B 5.8308,C 0.1652,E1 5.962,E2 414.2352} C_DIS
LIN {X 109.8834,Y 87.3989,Z 178,A 40.8042,B 5.8311,C 0.1561,E1 5.9577,E2 411.6847} C_DIS
LIN {X 107.4749,Y 90.3449,Z 178,A 41.8485,B 5.831,C 0.1606,E1 5.9559,E2 410.7055} C_DIS
LIN {X 105.2713,Y 92.9032,Z 178,A 43.4266,B 5.8311,C 0.1545,E1 5.953,E2 409.1013} C_DIS
LIN {X 102.2004,Y 96.2711,Z 178,A 45.2465,B 5.8312,C 0.1512,E1 5.9495,E2 407.2861} C_DIS
LIN {X 98.8957,Y 99.6628,Z 178,A 47.3648,B 5.8314,C 0.1444,E1 5.9453,E2 405.1433} C_DIS
LIN {X 96.3711,Y 102.1056,Z 178,A 48.8052,B 5.8314,C 0.1415,E1 5.9424,E2 403.7018} C_DIS
LIN {X 93.6202,Y 104.6341,Z 178,A 49.7708,B 5.8314,C 0.1471,E1 5.9405,E2 402.8078} C_DIS
LIN {X 91.2615,Y 106.6984,Z 178,A 51.3499,B 5.8314,C 0.1402,E1 5.9371,E2 401.1901} C_DIS
LIN {X 88.0479,Y 109.3646,Z 178,A 52.9442,B 5.8315,C 0.1387,E1 5.9337,E2 399.6096} C_DIS
LIN {X 84.6112,Y 112.0445,Z 178,A 54.7265,B 5.8315,C 0.1356,E1 5.9297,E2 397.8265} C_DIS
LIN {X 80.9154,Y 114.742,Z 178,A 56.8201,B 5.8317,C 0.1291,E1 5.9249,E2 395.7038} C_DIS
LIN {X 77.9183,Y 116.7979,Z 178,A 57.879,B 5.8317,C 0.133,E1 5.9226,E2 394.6992} C_DIS
LIN {X 74.7288,Y 118.8642,Z 178,A 59.5899,B 5.8317,C 0.1282,E1 5.9185,E2 392.9678} C_DIS
LIN {X 70.7109,Y 121.2979,Z 178,A 61.4683,B 5.8318,C 0.1259,E1 5.914,E2 391.0942} C_DIS
LIN {X 66.8027,Y 123.4933,Z 178,A 63.2895,B 5.8318,C 0.1235,E1 5.9095,E2 389.2741} C_DIS
LIN {X 62.6815,Y 125.6339,Z 178,A 65.256,B 5.8319,C 0.12,E1 5.9046,E2 387.2986} C_DIS
LIN {X 58.8167,Y 127.4875,Z 178,A 66.796,B 5.8319,C 0.1208,E1 5.9008,E2 385.7854} C_DIS
LIN {X 55.0368,Y 129.1665,Z 178,A 68.4103,B 5.8319,C 0.1199,E1 5.8967,E2 384.1807} C_DIS
LIN {X 50.6932,Y 130.9302,Z 178,A 70.321,B 5.8319,C 0.1179,E1 5.8917,E2 382.2705} C_DIS
LIN {X 47.1791,Y 132.2378,Z 178,A 71.9414,B 5.832,C 0.1151,E1 5.8874,E2 380.6388} C_DIS
LIN {X 44.0034,Y 133.328,Z 178,A 73.2122,B 5.832,C 0.1151,E1 5.8841,E2 379.3809} C_DIS
LIN {X 40.8897,Y 134.3152,Z 178,A 74.5417,B 5.832,C 0.1141,E1 5.8806,E2 378.052} C_DIS
LIN {X 37.4235,Y 135.3224,Z 178,A 76.0305,B 5.832,C 0.1127,E1 5.8766,E2 376.5615} C_DIS
LIN {X 30.8164,Y 136.9785,Z 178,A 78.7839,B 5.8321,C 0.1111,E1 5.8691,E2 373.8123} C_DIS
LIN {X 27.1417,Y 137.7552,Z 178,A 80.2738,B 5.8321,C 0.1108,E1 5.865,E2 372.3283} C_DIS
LIN {X 23.9414,Y 138.3474,Z 178,A 81.6027,B 5.8321,C 0.11,E1 5.8614,E2 370.9997} C_DIS
LIN {X 17.6868,Y 139.2841,Z 178,A 84.1441,B 5.8321,C 0.1095,E1 5.8544,E2 368.4642} C_DIS
LIN {X 14.6291,Y 139.6378,Z 178,A 85.4894,B 5.8321,C 0.1078,E1 5.8506,E2 367.1081} C_DIS
LIN {X 10.2764,Y 140.025,Z 178,A 87.2911,B 5.8321,C 0.1071,E1 5.8456,E2 365.3047} C_DIS
LIN {X 5.5385,Y 140.2924,Z 178,A 89.2189,B 5.8321,C 0.1069,E1 5.8402,E2 363.3788} C_DIS
LIN {X 1.3367,Y 140.3964,Z 178,A 90.9562,B 5.8321,C 0.1065,E1 5.8354,E2 361.6394} C_DIS
LIN {X -2.5628,Y 140.3785,Z 178,A 92.4939,B 5.8321,C 0.1072,E1 5.8311,E2 360.1092} C_DIS
LIN {X -6.5188,Y 140.2512,Z 178,A 94.1199,B 5.8321,C 0.1072,E1 5.8265,E2 358.4827} C_DIS
LIN {X -10.6049,Y 140.001,Z 178,A 96.0493,B 5.8322,C 0.1042,E1 5.8211,E2 356.5212} C_DIS
LIN {X -14.0611,Y 139.6972,Z 178,A 97.2382,B 5.8322,C 0.1074,E1 5.8178,E2 355.3619} C_DIS
LIN {X -17.9942,Y 139.2438,Z 178,A 98.8195,B 5.8322,C 0.1083,E1 5.8135,E2 353.7858} C_DIS
LIN {X -24.0468,Y 138.3278,Z 178,A 101.3659,B 5.8322,C 0.1088,E1 5.8064,E2 351.2347} C_DIS
LIN {X -29.4717,Y 137.2734,Z 178,A 103.3035,B 5.832,C 0.1139,E1 5.8013,E2 349.3386} C_DIS
LIN {X -33.2944,Y 136.3971,Z 178,A 105.3085,B 5.8321,C 0.1099,E1 5.7957,E2 347.2835} C_DIS
LIN {X -38.5543,Y 135.0062,Z 178,A 107.3985,B 5.8321,C 0.1131,E1 5.7901,E2 345.2114} C_DIS
LIN {X -41.2405,Y 134.2079,Z 178,A 108.5485,B 5.8321,C 0.114,E1 5.787,E2 344.0612} C_DIS
LIN {X -44.8682,Y 133.04,Z 178,A 110.1308,B 5.8321,C 0.115,E1 5.7828,E2 342.4766} C_DIS
LIN {X -48.5389,Y 131.7461,Z 178,A 112.085,B 5.8321,C 0.1122,E1 5.7775,E2 340.4771} C_DIS
LIN {X -51.9409,Y 130.4415,Z 178,A 113.1248,B 5.8319,C 0.119,E1 5.775,E2 339.495} C_DIS
LIN {X -54.6704,Y 129.3213,Z 178,A 114.4332,B 5.8319,C 0.119,E1 5.7716,E2 338.1743} C_DIS
LIN {X -57.8347,Y 127.9372,Z 178,A 115.9252,B 5.8319,C 0.1197,E1 5.7678,E2 336.6728} C_DIS
LIN {X -62.9543,Y 125.4986,Z 178,A 118.1908,B 5.8319,C 0.1231,E1 5.7621,E2 334.4151} C_DIS
LIN {X -65.4011,Y 124.2384,Z 178,A 119.3165,B 5.8319,C 0.1245,E1 5.7593,E2 333.2899} C_DIS
LIN {X -68.9417,Y 122.3115,Z 178,A 121.0769,B 5.8319,C 0.1254,E1 5.755,E2 331.5162} C_DIS
LIN {X -72.7842,Y 120.0646,Z 178,A 122.9018,B 5.8318,C 0.1279,E1 5.7506,E2 329.6916} C_DIS
LIN {X -76.5314,Y 117.7115,Z 178,A 124.7542,B 5.8318,C 0.1302,E1 5.7462,E2 327.8347} C_DIS
LIN {X -80.2674,Y 115.1963,Z 178,A 126.7066,B 5.8317,C 0.1318,E1 5.7417,E2 325.8692} C_DIS
LIN {X -85.7075,Y 111.2088,Z 178,A 129.2315,B 5.8315,C 0.139,E1 5.7361,E2 323.3755} C_DIS
LIN {X -89.1291,Y 108.4857,Z 178,A 131.1532,B 5.8315,C 0.1407,E1 5.7319,E2 321.4379} C_DIS
LIN {X -95.3427,Y 103.0678,Z 178,A 134.8283,B 5.8314,C 0.1436,E1 5.7241,E2 317.7263} C_DIS
LIN {X -100.3847,Y 98.1631,Z 178,A 138.387,B 5.8314,C 0.1419,E1 5.717,E2 314.0816} C_DIS
LIN {X -104.9039,Y 93.3185,Z 178,A 140.7994,B 5.8312,C 0.1508,E1 5.7125,E2 311.7092} C_DIS
LIN {X -107.9925,Y 89.7256,Z 178,A 142.0475,B 5.8309,C 0.1623,E1 5.7105,E2 310.5504} C_DIS
LIN {X -109.9762,Y 87.2829,Z 178,A 143.7471,B 5.8309,C 0.1608,E1 5.7074,E2 308.799} C_DIS
LIN {X -113.0879,Y 83.2115,Z 178,A 145.7281,B 5.8308,C 0.1667,E1 5.7041,E2 306.8339} C_DIS
LIN {X -115.5554,Y 79.7503,Z 178,A 147.5049,B 5.8307,C 0.1704,E1 5.7013,E2 305.0534} C_DIS
LIN {X -117.9877,Y 76.1059,Z 178,A 149.3226,B 5.8306,C 0.1743,E1 5.6985,E2 303.2335} C_DIS
LIN {X -120.2782,Y 72.4309,Z 178,A 151.1541,B 5.8305,C 0.178,E1 5.6958,E2 301.3953} C_DIS
LIN {X -122.4548,Y 68.6866,Z 178,A 152.9551,B 5.8303,C 0.182,E1 5.6933,E2 299.5916} C_DIS
LIN {X -126.2675,Y 61.3972,Z 178,A 156.3385,B 5.8301,C 0.1903,E1 5.689,E2 296.2079} C_DIS
LIN {X -128.3085,Y 57.0046,Z 178,A 158.1687,B 5.8298,C 0.1969,E1 5.6869,E2 294.3982} C_DIS
LIN {X -129.5279,Y 54.1756,Z 178,A 160.0097,B 5.8299,C 0.1943,E1 5.6848,E2 292.4833} C_DIS
LIN {X -130.9946,Y 50.5275,Z 178,A 161.0716,B 5.8296,C 0.2041,E1 5.6838,E2 291.4926} C_DIS
LIN {X -132.0787,Y 47.6206,Z 178,A 162.616,B 5.8296,C 0.2046,E1 5.6823,E2 289.9136} C_DIS
LIN {X -133.5023,Y 43.4771,Z 178,A 164.3555,B 5.8294,C 0.21,E1 5.6807,E2 288.1821} C_DIS
LIN {X -134.7046,Y 39.5878,Z 178,A 166.1137,B 5.8293,C 0.2136,E1 5.6793,E2 286.4127} C_DIS
LIN {X -135.8394,Y 35.5057,Z 178,A 167.8261,B 5.8291,C 0.2185,E1 5.6781,E2 284.704} C_DIS
LIN {X -136.6227,Y 32.3587,Z 178,A 169.2002,B 5.829,C 0.2217,E1 5.6772,E2 283.3245} C_DIS
LIN {X -137.2965,Y 29.3646,Z 178,A 170.5442,B 5.8289,C 0.2242,E1 5.6763,E2 281.9697} C_DIS
LIN {X -138.4726,Y 23.1928,Z 178,A 172.8614,B 5.8285,C 0.2339,E1 5.6752,E2 279.6866} C_DIS
LIN {X -139.0932,Y 19.1362,Z 178,A 174.9506,B 5.8285,C 0.2345,E1 5.6743,E2 277.5455} C_DIS
LIN {X -140.0189,Y 10.36,Z 178,A 178.5055,B 5.828,C 0.2453,E1 5.6734,E2 273.9997} C_DIS
LIN {X -140.3466,Y 3.9323,Z 178,A -179.0831,B 5.8276,C 0.2549,E1 5.6731,E2 271.6182} C_DIS
LIN {X -140.363,Y -3.3422,Z 178,A -175.4445,B 5.8276,C 0.2567,E1 5.6731,E2 267.8955} C_DIS
LIN {X -140.0063,Y -10.5321,Z 178,A -171.8607,B 5.8274,C 0.2585,E1 5.6738,E2 264.2291} C_DIS
LIN {X -139.3895,Y -16.8284,Z 178,A -169.6555,B 5.8269,C 0.2696,E1 5.6745,E2 262.0753} C_DIS
LIN {X -138.848,Y -20.8376,Z 178,A -168.4324,B 5.8265,C 0.2786,E1 5.6749,E2 260.9094} C_DIS
LIN {X -138.2651,Y -24.4016,Z 178,A -166.7667,B 5.8265,C 0.2808,E1 5.6757,E2 259.2196} C_DIS
LIN {X -137.5066,Y -28.3657,Z 178,A -165.1053,B 5.8262,C 0.2852,E1 5.6766,E2 257.5575} C_DIS
LIN {X -136.6351,Y -32.3072,Z 178,A -163.4006,B 5.826,C 0.2892,E1 5.6777,E2 255.8464} C_DIS
LIN {X -135.64,Y -36.2537,Z 178,A -161.7646,B 5.8258,C 0.294,E1 5.6788,E2 254.2146} C_DIS
LIN {X -134.5042,Y -40.2722,Z 178,A -160.0476,B 5.8255,C 0.2985,E1 5.6802,E2 252.4972} C_DIS
LIN {X -133.7026,Y -42.8502,Z 178,A -158.8682,B 5.8255,C 0.3007,E1 5.6812,E2 251.3082} C_DIS
LIN {X -132.5097,Y -46.4099,Z 178,A -156.7203,B 5.8255,C 0.2984,E1 5.6832,E2 249.0802} C_DIS
LIN {X -130.7445,Y -51.171,Z 178,A -154.9252,B 5.8251,C 0.3067,E1 5.685,E2 247.3228} C_DIS
LIN {X -129.5016,Y -54.2385,Z 178,A -153.8483,B 5.8248,C 0.3131,E1 5.6861,E2 246.2827} C_DIS
LIN {X -128.0656,Y -57.5477,Z 178,A -152.2875,B 5.8246,C 0.316,E1 5.6879,E2 244.711} C_DIS
LIN {X -126.5618,Y -60.7837,Z 178,A -150.8231,B 5.8244,C 0.3196,E1 5.6897,E2 243.2463} C_DIS
LIN {X -124.8687,Y -64.1916,Z 178,A -149.2716,B 5.8242,C 0.3235,E1 5.6916,E2 241.6957} C_DIS
LIN {X -120.0359,Y -72.8317,Z 178,A -145.0759,B 5.8237,C 0.3318,E1 5.6974,E2 237.4818} C_DIS
LIN {X -117.2358,Y -77.2579,Z 178,A -142.8564,B 5.8235,C 0.3359,E1 5.7008,E2 235.2523} C_DIS
LIN {X -114.6666,Y -81.0223,Z 178,A -140.9814,B 5.8233,C 0.34,E1 5.7038,E2 233.3761} C_DIS
LIN {X -112.0846,Y -84.558,Z 178,A -139.1405,B 5.8231,C 0.3434,E1 5.7069,E2 231.5287} C_DIS
LIN {X -109.2691,Y -88.1662,Z 178,A -137.2403,B 5.8229,C 0.3471,E1 5.7102,E2 229.6247} C_DIS
LIN {X -106.3781,Y -91.6337,Z 178,A -135.3476,B 5.8227,C 0.3504,E1 5.7136,E2 227.7259} C_DIS
LIN {X -103.338,Y -95.0488,Z 178,A -133.4732,B 5.8224,C 0.3541,E1 5.7171,E2 225.8509} C_DIS
LIN {X -100.296,Y -98.2534,Z 178,A -131.636,B 5.8222,C 0.3573,E1 5.7207,E2 224.0097} C_DIS
LIN {X -97.1551,Y -101.3605,Z 178,A -129.7849,B 5.8221,C 0.3602,E1 5.7244,E2 222.1526} C_DIS
LIN {X -93.9068,Y -104.3774,Z 178,A -127.9199,B 5.8219,C 0.3629,E1 5.7282,E2 220.2804} C_DIS
LIN {X -90.4916,Y -107.3517,Z 178,A -126.0893,B 5.8217,C 0.3664,E1 5.7321,E2 218.4524} C_DIS
LIN {X -87.2274,Y -110.0204,Z 178,A -124.3252,B 5.8215,C 0.3688,E1 5.736,E2 216.6828} C_DIS
LIN {X -83.5539,Y -112.8357,Z 178,A -122.3281,B 5.8215,C 0.3707,E1 5.7405,E2 214.6714} C_DIS
LIN {X -79.9892,Y -115.3898,Z 178,A -120.6614,B 5.8211,C 0.3749,E1 5.7442,E2 213.0213} C_DIS
LIN {X -76.6336,Y -117.6451,Z 178,A -118.8598,B 5.8211,C 0.3755,E1 5.7485,E2 211.1996} C_DIS
LIN {X -72.4872,Y -120.2442,Z 178,A -116.8991,B 5.8209,C 0.3787,E1 5.7531,E2 209.2437} C_DIS
LIN {X -68.5857,Y -122.5116,Z 178,A -115.0744,B 5.8207,C 0.3814,E1 5.7576,E2 207.4212} C_DIS
LIN {X -64.978,Y -124.4605,Z 178,A -113.1977,B 5.8207,C 0.3809,E1 5.7623,E2 205.5172} C_DIS
LIN {X -61.622,Y -126.1566,Z 178,A -111.8837,B 5.8205,C 0.3854,E1 5.7655,E2 204.2326} C_DIS
LIN {X -58.2194,Y -127.7637,Z 178,A -110.1146,B 5.8205,C 0.3842,E1 5.77,E2 202.4323} C_DIS
LIN {X -53.9018,Y -129.6423,Z 178,A -108.4117,B 5.8202,C 0.3889,E1 5.7743,E2 200.7582} C_DIS
LIN {X -50.3212,Y -131.0748,Z 178,A -106.8205,B 5.8202,C 0.3901,E1 5.7785,E2 199.1645} C_DIS
LIN {X -47.2357,Y -132.2174,Z 178,A -105.4591,B 5.8201,C 0.391,E1 5.7821,E2 197.8004} C_DIS
LIN {X -44.1224,Y -133.2883,Z 178,A -104.0991,B 5.8201,C 0.3919,E1 5.7857,E2 196.4379} C_DIS
LIN {X -40.5141,Y -134.4302,Z 178,A -102.5154,B 5.82,C 0.3925,E1 5.7899,E2 194.8487} C_DIS
LIN {X -34.3662,Y -136.1305,Z 178,A -99.9376,B 5.8198,C 0.3945,E1 5.7969,E2 192.2736} C_DIS
LIN {X -30.7825,Y -136.9862,Z 178,A -98.4227,B 5.8198,C 0.3951,E1 5.801,E2 190.7568} C_DIS
LIN {X -27.2619,Y -137.7312,Z 178,A -96.9229,B 5.8198,C 0.3954,E1 5.8051,E2 189.2525} C_DIS
LIN {X -22.1395,Y -138.6465,Z 178,A -94.7477,B 5.8198,C 0.3954,E1 5.8111,E2 187.0697} C_DIS
LIN {X -18.4298,Y -139.1867,Z 178,A -93.2024,B 5.8198,C 0.3957,E1 5.8154,E2 185.5216} C_DIS
LIN {X -14.8148,Y -139.6179,Z 178,A -91.8173,B 5.8197,C 0.3973,E1 5.8192,E2 184.1495} C_DIS
LIN {X -11.3495,Y -139.9429,Z 178,A -90.3801,B 5.8197,C 0.3973,E1 5.8232,E2 182.7095} C_DIS
LIN {X -7.0774,Y -140.2231,Z 178,A -88.5568,B 5.8197,C 0.3963,E1 5.8283,E2 180.8752} C_DIS
LIN {X -3.1943,Y -140.3671,Z 178,A -86.9002,B 5.8197,C 0.3953,E1 5.833,E2 179.2084} C_DIS
LIN {X 1.0219,Y -140.3968,Z 178,A -85.9441,B 5.8191,C 0.4055,E1 5.8354,E2 178.3537} C_DIS
Enddeposition()
LIN {X 1.0219,Y -140.3968,Z 178,A -85.9441,B 5.8191,C 0.4055,E1 5.8354,E2 178.3537} C_DIS
Startdeposition()
$VEL.CP = VEL_PRINT
LIN {X -0.22,Y -141.3068,Z 178,A -86.389,B 5.8189,C 0.4081,E1 5.8341,E2 178.8238} C_DIS
LIN {X -3.876,Y -141.2527,Z 178,A -87.9319,B 5.8189,C 0.409,E1 5.8297,E2 180.3755} C_DIS
LIN {X -8.2031,Y -141.0683,Z 178,A -89.6197,B 5.8189,C 0.4081,E1 5.825,E2 182.055} C_DIS
LIN {X -11.288,Y -140.8555,Z 178,A -90.8443,B 5.8189,C 0.4076,E1 5.8216,E2 183.2762} C_DIS
LIN {X -14.1215,Y -140.5997,Z 178,A -92.0392,B 5.8189,C 0.408,E1 5.8183,E2 184.477} C_DIS
LIN {X -17.2529,Y -140.2495,Z 178,A -93.4934,B 5.8188,C 0.41,E1 5.8142,E2 185.9553} C_DIS
LIN {X -21.4025,Y -139.6756,Z 178,A -95.0081,B 5.819,C 0.4071,E1 5.8101,E2 187.446} C_DIS
LIN {X -25.4445,Y -138.997,Z 178,A -96.7846,B 5.819,C 0.408,E1 5.8051,E2 189.2384} C_DIS
LIN {X -29.0429,Y -138.291,Z 178,A -98.3866,B 5.8189,C 0.4088,E1 5.8007,E2 190.8563} C_DIS
LIN {X -32.6838,Y -137.4744,Z 178,A -99.762,B 5.819,C 0.4062,E1 5.797,E2 192.2137} C_DIS
LIN {X -35.7522,Y -136.7095,Z 178,A -101.1239,B 5.819,C 0.4065,E1 5.7933,E2 193.5866} C_DIS
LIN {X -40.4627,Y -135.3906,Z 178,A -103.0292,B 5.8192,C 0.4042,E1 5.7882,E2 195.4819} C_DIS
LIN {X -43.8415,Y -134.3349,Z 178,A -104.6743,B 5.8191,C 0.4057,E1 5.7838,E2 197.1553} C_DIS
LIN {X -47.931,Y -132.9279,Z 178,A -106.4012,B 5.8191,C 0.4039,E1 5.7792,E2 198.8788} C_DIS
LIN {X -52.3671,Y -131.2446,Z 178,A -108.1217,B 5.8195,C 0.3996,E1 5.7748,E2 200.5726} C_DIS
LIN {X -55.594,Y -129.9107,Z 178,A -109.4689,B 5.8196,C 0.3974,E1 5.7714,E2 201.9108} C_DIS
LIN {X -58.5034,Y -128.6284,Z 178,A -111.0585,B 5.8195,C 0.3997,E1 5.7672,E2 203.5406} C_DIS
LIN {X -62.5881,Y -126.6883,Z 178,A -112.7533,B 5.8197,C 0.3959,E1 5.763,E2 205.2171} C_DIS
LIN {X -66.2614,Y -124.8079,Z 178,A -114.4836,B 5.8198,C 0.3946,E1 5.7587,E2 206.955} C_DIS
LIN {X -70.2515,Y -122.6073,Z 178,A -116.4093,B 5.8199,C 0.3931,E1 5.754,E2 208.8912} C_DIS
LIN {X -74.251,Y -120.2278,Z 178,A -118.2497,B 5.8201,C 0.39,E1 5.7496,E2 210.7254} C_DIS
LIN {X -77.9131,Y -117.8871,Z 178,A -120.0186,B 5.8203,C 0.3875,E1 5.7454,E2 212.4951} C_DIS
LIN {X -81.0207,Y -115.7737,Z 178,A -121.5362,B 5.8205,C 0.3851,E1 5.742,E2 214.0118} C_DIS
LIN {X -83.9929,Y -113.6359,Z 178,A -123.1586,B 5.8205,C 0.3843,E1 5.7383,E2 215.6523} C_DIS
LIN {X -87.6125,Y -110.8692,Z 178,A -125.0464,B 5.8207,C 0.3817,E1 5.7341,E2 217.5453} C_DIS
LIN {X -91.1228,Y -108.0025,Z 178,A -126.8972,B 5.8209,C 0.3787,E1 5.7301,E2 219.3975} C_DIS
LIN {X -94.571,Y -104.9963,Z 178,A -128.7651,B 5.8211,C 0.3755,E1 5.7262,E2 221.2668} C_DIS
LIN {X -97.8051,Y -101.9901,Z 178,A -130.576,B 5.8213,C 0.3723,E1 5.7225,E2 223.08} C_DIS
LIN {X -100.8506,Y -98.9793,Z 178,A -132.3336,B 5.8215,C 0.3692,E1 5.719,E2 224.8401} C_DIS
LIN {X -103.7799,Y -95.9042,Z 178,A -134.1101,B 5.8217,C 0.3663,E1 5.7156,E2 226.6233} C_DIS
LIN {X -106.7623,Y -92.573,Z 178,A -135.9849,B 5.8219,C 0.3633,E1 5.7122,E2 228.5057} C_DIS
LIN {X -109.7331,Y -89.0313,Z 178,A -137.864,B 5.8221,C 0.3593,E1 5.7088,E2 230.3848} C_DIS
LIN {X -112.4836,Y -85.5298,Z 178,A -139.7124,B 5.8223,C 0.3558,E1 5.7056,E2 232.2383} C_DIS
LIN {X -115.1432,Y -81.914,Z 178,A -141.5729,B 5.8225,C 0.3521,E1 5.7026,E2 234.1035} C_DIS
LIN {X -117.7141,Y -78.1745,Z 178,A -143.1958,B 5.8229,C 0.3455,E1 5.7001,E2 235.697} C_DIS
LIN {X -119.5738,Y -75.2986,Z 178,A -144.8079,B 5.8229,C 0.3447,E1 5.6976,E2 237.338} C_DIS
LIN {X -121.7433,Y -71.7381,Z 178,A -146.4275,B 5.8233,C 0.3399,E1 5.6953,E2 238.9475} C_DIS
LIN {X -124.8611,Y -66.1602,Z 178,A -149.1143,B 5.8236,C 0.3345,E1 5.6917,E2 241.6457} C_DIS
LIN {X -126.5622,Y -62.8437,Z 178,A -150.6868,B 5.8238,C 0.3314,E1 5.6897,E2 243.2255} C_DIS
LIN {X -128.0188,Y -59.8222,Z 178,A -151.9641,B 5.824,C 0.327,E1 5.6881,E2 244.4913} C_DIS
LIN {X -129.4873,Y -56.5733,Z 178,A -153.6438,B 5.824,C 0.3258,E1 5.6862,E2 246.2008} C_DIS
LIN {X -130.7822,Y -53.5143,Z 178,A -155.8983,B 5.8237,C 0.3316,E1 5.6838,E2 248.5722} C_DIS
LIN {X -133.2677,Y -46.9838,Z 178,A -157.8857,B 5.8246,C 0.3154,E1 5.6819,E2 250.4487} C_DIS
LIN {X -134.3382,Y -43.8314,Z 178,A -159.3938,B 5.8248,C 0.3134,E1 5.6806,E2 251.9766} C_DIS
LIN {X -135.6507,Y -39.5746,Z 178,A -160.9963,B 5.8251,C 0.3064,E1 5.6793,E2 253.5514} C_DIS
LIN {X -136.4291,Y -36.8036,Z 178,A -162.2467,B 5.8252,C 0.3041,E1 5.6784,E2 254.8119} C_DIS
LIN {X -137.2563,Y -33.5887,Z 178,A -163.6227,B 5.8254,C 0.3007,E1 5.6775,E2 256.1909} C_DIS
LIN {X -137.9657,Y -30.5496,Z 178,A -164.9246,B 5.8256,C 0.2976,E1 5.6766,E2 257.4968} C_DIS
LIN {X -138.6062,Y -27.497,Z 178,A -166.21,B 5.8257,C 0.2943,E1 5.6759,E2 258.784} C_DIS
LIN {X -139.2956,Y -23.7545,Z 178,A -167.6806,B 5.826,C 0.2892,E1 5.6752,E2 260.2441} C_DIS
LIN {X -139.8549,Y -20.198,Z 178,A -169.4215,B 5.826,C 0.2879,E1 5.6745,E2 262.0205} C_DIS
LIN {X -140.397,Y -16.0146,Z 178,A -171.611,B 5.826,C 0.2879,E1 5.6737,E2 264.2705} C_DIS
LIN {X -140.8474,Y -11.3837,Z 178,A -172.9829,B 5.8266,C 0.2774,E1 5.6734,E2 265.5748} C_DIS
LIN {X -141.0924,Y -7.7948,Z 178,A -174.5808,B 5.8266,C 0.2747,E1 5.6731,E2 267.1896} C_DIS
LIN {X -141.2277,Y -4.7577,Z 178,A -176.0218,B 5.8268,C 0.2732,E1 5.6731,E2 268.6565} C_DIS
LIN {X -141.3,Y 1.4729,Z 178,A -178.4478,B 5.8271,C 0.265,E1 5.673,E2 271.0676} C_DIS
LIN {X -141.2097,Y 5.2189,Z 178,A -179.9607,B 5.8273,C 0.2606,E1 5.6731,E2 272.5785} C_DIS
LIN {X -140.9985,Y 9.3372,Z 178,A 178.4185,B 5.8276,C 0.2553,E1 5.6734,E2 274.1913} C_DIS
LIN {X -140.7123,Y 12.9487,Z 178,A 176.3683,B 5.8276,C 0.2569,E1 5.6739,E2 276.3149} C_DIS
LIN {X -140.2314,Y 17.4041,Z 178,A 174.9029,B 5.8279,C 0.2483,E1 5.6744,E2 277.7338} C_DIS
LIN {X -139.7531,Y 20.9016,Z 178,A 173.3471,B 5.8279,C 0.2455,E1 5.675,E2 279.3044} C_DIS
LIN {X -138.2001,Y 29.4639,Z 178,A 169.8829,B 5.8284,C 0.2349,E1 5.6768,E2 282.7573} C_DIS
LIN {X -137.4147,Y 32.9316,Z 178,A 168.4591,B 5.8286,C 0.2307,E1 5.6777,E2 284.1775} C_DIS
LIN {X -136.6799,Y 35.8634,Z 178,A 167.2211,B 5.8287,C 0.2275,E1 5.6786,E2 285.4161} C_DIS
LIN {X -135.8884,Y 38.7572,Z 178,A 165.9525,B 5.8288,C 0.2246,E1 5.6795,E2 286.6904} C_DIS
LIN {X -134.739,Y 42.5774,Z 178,A 164.2494,B 5.829,C 0.2211,E1 5.6809,E2 288.403} C_DIS
LIN {X -133.6248,Y 45.9539,Z 178,A 162.7192,B 5.829,C 0.218,E1 5.6823,E2 289.9432} C_DIS
LIN {X -132.0281,Y 50.364,Z 178,A 160.8591,B 5.8293,C 0.2125,E1 5.6841,E2 291.7964} C_DIS
LIN {X -130.0455,Y 55.2821,Z 178,A 158.5097,B 5.8294,C 0.2089,E1 5.6866,E2 294.1694} C_DIS
LIN {X -128.4097,Y 58.9769,Z 178,A 157.0759,B 5.8296,C 0.2025,E1 5.6882,E2 295.5755} C_DIS
LIN {X -127.2966,Y 61.3432,Z 178,A 155.596,B 5.8296,C 0.204,E1 5.6901,E2 297.1079} C_DIS
LIN {X -125.8223,Y 64.3116,Z 178,A 154.2702,B 5.8297,C 0.2004,E1 5.6918,E2 298.4301} C_DIS
LIN {X -124.281,Y 67.2471,Z 178,A 153.0803,B 5.8299,C 0.1955,E1 5.6933,E2 299.5993} C_DIS
LIN {X -122.2149,Y 70.9316,Z 178,A 151.3097,B 5.83,C 0.1918,E1 5.6958,E2 301.3757} C_DIS
LIN {X -119.8701,Y 74.8262,Z 178,A 149.4268,B 5.8301,C 0.1877,E1 5.6985,E2 303.262} C_DIS
LIN {X -117.3365,Y 78.7402,Z 178,A 147.5684,B 5.8303,C 0.1829,E1 5.7013,E2 305.1146} C_DIS
LIN {X -114.9435,Y 82.1933,Z 178,A 145.8071,B 5.8303,C 0.1795,E1 5.7042,E2 306.8818} C_DIS
LIN {X -110.3927,Y 88.2116,Z 178,A 142.8204,B 5.8306,C 0.1718,E1 5.7092,E2 309.8567} C_DIS
LIN {X -106.1578,Y 93.2656,Z 178,A 139.8501,B 5.8307,C 0.1692,E1 5.7147,E2 312.8623} C_DIS
LIN {X -101.4588,Y 98.3558,Z 178,A 137.0704,B 5.8309,C 0.163,E1 5.72,E2 315.6358} C_DIS
LIN {X -98.3073,Y 101.5058,Z 178,A 135.2302,B 5.8309,C 0.1598,E1 5.7236,E2 317.4787} C_DIS
LIN {X -94.2912,Y 105.247,Z 178,A 132.5748,B 5.8309,C 0.1601,E1 5.7292,E2 320.1864} C_DIS
LIN {X -91.0768,Y 108.0411,Z 178,A 131.1804,B 5.8311,C 0.1534,E1 5.7321,E2 321.5375} C_DIS
LIN {X -87.5676,Y 110.9045,Z 178,A 129.3197,B 5.8312,C 0.1504,E1 5.7361,E2 323.3997} C_DIS
LIN {X -80.8986,Y 115.8586,Z 178,A 125.8767,B 5.8313,C 0.1456,E1 5.7439,E2 326.8494} C_DIS
LIN {X -76.9667,Y 118.5069,Z 178,A 123.9604,B 5.8314,C 0.1425,E1 5.7484,E2 328.7635} C_DIS
LIN {X -73.0586,Y 120.9554,Z 178,A 122.0426,B 5.8314,C 0.1403,E1 5.753,E2 330.6858} C_DIS
LIN {X -68.9403,Y 123.3496,Z 178,A 120.0815,B 5.8315,C 0.1379,E1 5.7577,E2 332.6491} C_DIS
LIN {X -64.8531,Y 125.5466,Z 178,A 118.3014,B 5.8316,C 0.1343,E1 5.7621,E2 334.4151} C_DIS
LIN {X -61.4759,Y 127.2332,Z 178,A 116.7069,B 5.8316,C 0.1331,E1 5.7661,E2 336.0165} C_DIS
LIN {X -58.1193,Y 128.8004,Z 178,A 115.1813,B 5.8316,C 0.1316,E1 5.77,E2 337.5439} C_DIS
LIN {X -55.2146,Y 130.0739,Z 178,A 113.7431,B 5.8316,C 0.132,E1 5.7737,E2 339.0005} C_DIS
LIN {X -50.5026,Y 131.9743,Z 178,A 111.6784,B 5.8317,C 0.13,E1 5.7791,E2 341.0643} C_DIS
LIN {X -46.3982,Y 133.4707,Z 178,A 110.1705,B 5.8318,C 0.1252,E1 5.7829,E2 342.5377} C_DIS
LIN {X -43.8314,Y 134.3382,Z 178,A 108.9576,B 5.8318,C 0.1256,E1 5.7862,E2 343.7645} C_DIS
LIN {X -40.1565,Y 135.4803,Z 178,A 107.2611,B 5.8318,C 0.126,E1 5.7908,E2 345.4769} C_DIS
LIN {X -33.3564,Y 137.3123,Z 178,A 104.5153,B 5.8318,C 0.1227,E1 5.7982,E2 348.2072} C_DIS
LIN {X -29.6435,Y 138.1614,Z 178,A 102.6995,B 5.8318,C 0.1251,E1 5.8032,E2 350.0562} C_DIS
LIN {X -22.4434,Y 139.513,Z 178,A 99.793,B 5.8318,C 0.1229,E1 5.8112,E2 352.953} C_DIS
LIN {X -17.6165,Y 140.2053,Z 178,A 98.0144,B 5.8319,C 0.1197,E1 5.816,E2 354.7056} C_DIS
LIN {X -15.0207,Y 140.5052,Z 178,A 96.9974,B 5.8319,C 0.1189,E1 5.8188,E2 355.7167} C_DIS
LIN {X -12.1863,Y 140.7796,Z 178,A 95.742,B 5.8319,C 0.1199,E1 5.8224,E2 356.9842} C_DIS
LIN {X -9.2595,Y 141.0033,Z 178,A 94.5221,B 5.8319,C 0.1201,E1 5.8258,E2 358.2072} C_DIS
LIN {X -5.6672,Y 141.1923,Z 178,A 93.3109,B 5.8319,C 0.1168,E1 5.8291,E2 359.3865} C_DIS
LIN {X -3.2741,Y 141.2694,Z 178,A 92.1801,B 5.8319,C 0.1188,E1 5.8323,E2 360.5371} C_DIS
LIN {X -0.0081,Y 141.308,Z 178,A 90.6577,B 5.8319,C 0.1214,E1 5.8366,E2 362.0839} C_DIS
LIN {X 3.8616,Y 141.2531,Z 178,A 89.2041,B 5.8319,C 0.12,E1 5.8406,E2 363.5222} C_DIS
LIN {X 8.2908,Y 141.0629,Z 178,A 87.3768,B 5.8319,C 0.1207,E1 5.8457,E2 365.3526} C_DIS
LIN {X 12.1567,Y 140.7821,Z 178,A 85.7876,B 5.8319,C 0.1213,E1 5.8501,E2 366.9434} C_DIS
LIN {X 16.4011,Y 140.3511,Z 178,A 84.2402,B 5.8319,C 0.1195,E1 5.8544,E2 368.4671} C_DIS
LIN {X 19.3431,Y 139.977,Z 178,A 82.8198,B 5.8319,C 0.1229,E1 5.8584,E2 369.9146} C_DIS
LIN {X 24.127,Y 139.2328,Z 178,A 81.0421,B 5.8319,C 0.1214,E1 5.8632,E2 371.6684} C_DIS
LIN {X 27.9503,Y 138.5139,Z 178,A 79.5652,B 5.8319,C 0.1209,E1 5.8672,E2 373.132} C_DIS
LIN {X 30.5265,Y 137.9707,Z 178,A 78.3914,B 5.8319,C 0.123,E1 5.8705,E2 374.3191} C_DIS
LIN {X 34.4043,Y 137.0537,Z 178,A 76.5733,B 5.8318,C 0.1269,E1 5.8755,E2 376.1622} C_DIS
LIN {X 38.972,Y 135.8271,Z 178,A 74.7271,B 5.8318,C 0.1275,E1 5.8804,E2 377.9991} C_DIS
LIN {X 43.2212,Y 134.5333,Z 178,A 73.0434,B 5.8318,C 0.1275,E1 5.8849,E2 379.6676} C_DIS
LIN {X 47.5363,Y 133.0703,Z 178,A 71.2656,B 5.8318,C 0.1282,E1 5.8895,E2 381.4362} C_DIS
LIN {X 50.6496,Y 131.9173,Z 178,A 69.8864,B 5.8318,C 0.1301,E1 5.8931,E2 382.8195} C_DIS
LIN {X 53.4922,Y 130.7911,Z 178,A 68.7049,B 5.8317,C 0.1306,E1 5.8962,E2 383.9935} C_DIS
LIN {X 55.9563,Y 129.754,Z 178,A 67.5713,B 5.8317,C 0.1326,E1 5.8991,E2 385.1331} C_DIS
LIN {X 59.5594,Y 128.1403,Z 178,A 65.9956,B 5.8317,C 0.1341,E1 5.9031,E2 386.7056} C_DIS
LIN {X 63.6871,Y 126.1402,Z 178,A 63.8133,B 5.8314,C 0.1411,E1 5.9087,E2 388.9285} C_DIS
LIN {X 67.2439,Y 124.2827,Z 178,A 62.4656,B 5.8314,C 0.1394,E1 5.9119,E2 390.241} C_DIS
LIN {X 71.3258,Y 121.9855,Z 178,A 60.6036,B 5.8314,C 0.1415,E1 5.9164,E2 392.0983} C_DIS
LIN {X 75.0735,Y 119.7159,Z 178,A 58.8982,B 5.8314,C 0.1432,E1 5.9204,E2 393.7947} C_DIS
LIN {X 78.4502,Y 117.5301,Z 178,A 57.4403,B 5.8314,C 0.1432,E1 5.9238,E2 395.2306} C_DIS
LIN {X 81.6494,Y 115.3308,Z 178,A 55.693,B 5.8313,C 0.1484,E1 5.9278,E2 397.0001} C_DIS
LIN {X 85.4059,Y 112.5776,Z 178,A 53.828,B 5.8312,C 0.1513,E1 5.932,E2 398.8623} C_DIS
LIN {X 89.1003,Y 109.6771,Z 178,A 52.0559,B 5.8312,C 0.1527,E1 5.9359,E2 400.6178} C_DIS
LIN {X 92.5638,Y 106.7703,Z 178,A 50.4026,B 5.8312,C 0.1534,E1 5.9393,E2 402.2484} C_DIS
LIN {X 99.3574,Y 100.4787,Z 178,A 46.4398,B 5.8308,C 0.164,E1 5.9475,E2 406.2388} C_DIS
LIN {X 102.6351,Y 97.128,Z 178,A 44.6036,B 5.8308,C 0.1669,E1 5.951,E2 408.0673} C_DIS
LIN {X 105.1027,Y 94.4522,Z 178,A 43.1359,B 5.8307,C 0.1699,E1 5.9538,E2 409.5343} C_DIS
LIN {X 107.2837,Y 91.9678,Z 178,A 40.7582,B 5.8301,C 0.1887,E1 5.9583,E2 412.0438} C_DIS
LIN {X 112.5622,Y 85.4263,Z 178,A 38.4653,B 5.8304,C 0.1792,E1 5.962,E2 414.1967} C_DIS
LIN {X 115.3565,Y 81.6129,Z 178,A 36.6019,B 5.8303,C 0.1828,E1 5.965,E2 416.0539} C_DIS
LIN {X 117.8093,Y 78.0313,Z 178,A 34.9246,B 5.8303,C 0.1857,E1 5.9676,E2 417.7213} C_DIS
LIN {X 119.9688,Y 74.6675,Z 178,A 33.3542,B 5.8301,C 0.1888,E1 5.9699,E2 419.286} C_DIS
LIN {X 122.0295,Y 71.2509,Z 178,A 31.9693,B 5.8301,C 0.1891,E1 5.9719,E2 420.6415} C_DIS
LIN {X 123.752,Y 68.215,Z 178,A 30.3341,B 5.8299,C 0.1961,E1 5.9742,E2 422.3058} C_DIS
LIN {X 125.7708,Y 64.4127,Z 178,A 28.6954,B 5.8298,C 0.1988,E1 5.9763,E2 423.9314} C_DIS
LIN {X 127.4584,Y 61.0045,Z 178,A 27.1653,B 5.8296,C 0.2026,E1 5.9781,E2 425.4607} C_DIS
LIN {X 129.0972,Y 57.4559,Z 178,A 25.6468,B 5.8296,C 0.2056,E1 5.9799,E2 426.9715} C_DIS
LIN {X 130.6821,Y 53.7584,Z 178,A 24.0766,B 5.8294,C 0.2089,E1 5.9816,E2 428.5348} C_DIS
LIN {X 132.1234,Y 50.1095,Z 178,A 22.5135,B 5.8293,C 0.2127,E1 5.9831,E2 430.0951} C_DIS
LIN {X 133.2758,Y 46.9606,Z 178,A 21.2295,B 5.8292,C 0.2151,E1 5.9843,E2 431.3702} C_DIS
LIN {X 134.3067,Y 43.926,Z 178,A 19.7493,B 5.829,C 0.2216,E1 5.9857,E2 432.8746} C_DIS
LIN {X 135.7282,Y 39.3097,Z 178,A 17.8927,B 5.8288,C 0.2253,E1 5.9871,E2 434.7191} C_DIS
LIN {X 136.9927,Y 34.6448,Z 178,A 16.1347,B 5.8288,C 0.2274,E1 5.9884,E2 436.4522} C_DIS
LIN {X 137.6333,Y 32.01,Z 178,A 15.1211,B 5.8287,C 0.229,E1 5.989,E2 437.4553} C_DIS
LIN {X 138.4366,Y 28.3301,Z 178,A 13.6249,B 5.8285,C 0.2328,E1 5.9899,E2 438.9486} C_DIS
LIN {X 138.9436,Y 25.7412,Z 178,A 12.3162,B 5.8282,C 0.2397,E1 5.9906,E2 440.2891} C_DIS
LIN {X 139.5614,Y 22.1403,Z 178,A 11.1505,B 5.8282,C 0.2387,E1 5.9911,E2 441.4148} C_DIS
LIN {X 139.9536,Y 19.507,Z 178,A 9.6667,B 5.8279,C 0.2483,E1 5.9917,E2 442.9519} C_DIS
LIN {X 140.4091,Y 15.9123,Z 178,A 8.5703,B 5.8279,C 0.2464,E1 5.9921,E2 444.001} C_DIS
Enddeposition()
END
